FUNCTION "Automatico_linea_1" : VOID	// FC 5
NAME : Auto_L1
VERSION : 0.1
BEGIN
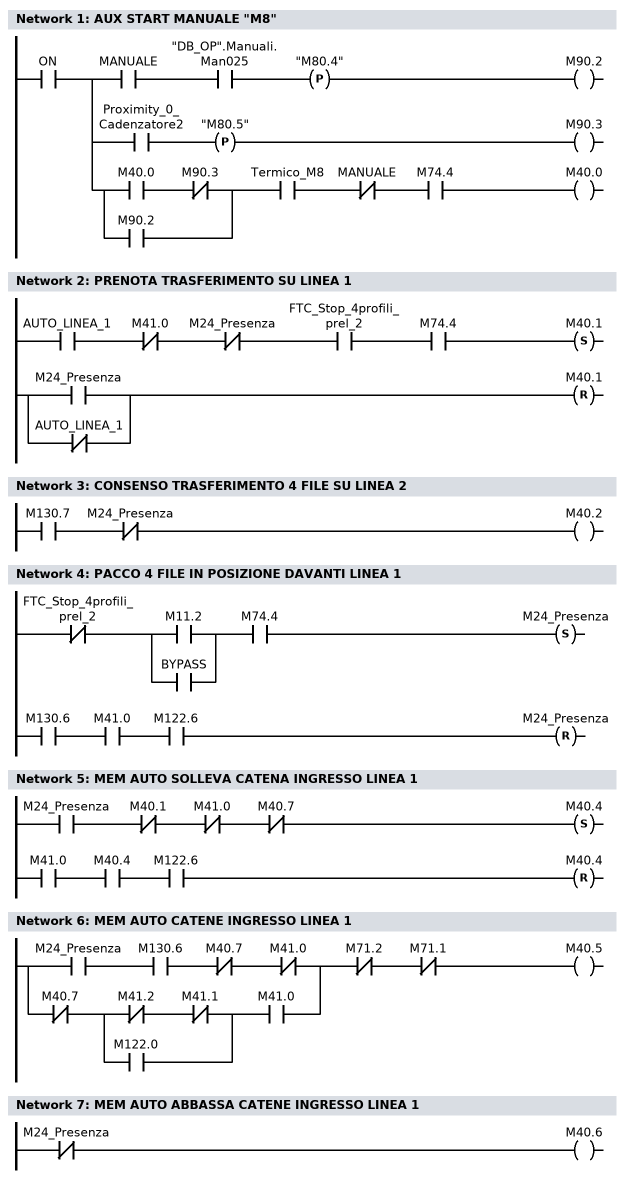
NETWORK
TITLE = AUX START MANUALE "M8"
      A     "ON";
      =     L 0.0;
      A     L 0.0;
      A     "MANUALE";
      A     "DB_OP".Manuali.Man025;
      FP    "M80.4";
      =     "M90.2";
      A     L 0.0;
      A     "Proximity_0_Cadenzatore2";
      FP    "M80.5";
      =     "M90.3";
      A     L 0.0;
      A(;
      A     "M40.0";
      AN    "M90.3";
      O     "M90.2";
      );
      A     "Termico_M8";
      AN    "MANUALE";
      A     "M74.4";
      =     "M40.0";
NETWORK
TITLE = PRENOTA TRASFERIMENTO SU LINEA 1
      A     "AUTO_LINEA_1";
      AN    "M41.0";
      AN    "M24_Presenza";
      A     "FTC_Stop_4profili_prel_2";
      A     "M74.4";
      S     "M40.1";
      A(;
      O     "M24_Presenza";
      ON    "AUTO_LINEA_1";
      );
      R     "M40.1";
      NOP   0;
NETWORK
TITLE = CONSENSO TRASFERIMENTO 4 FILE SU LINEA 2
      A     "M130.7";
      AN    "M24_Presenza";
      =     "M40.2";
NETWORK
TITLE = PACCO 4 FILE IN POSIZIONE DAVANTI LINEA 1
      AN    "FTC_Stop_4profili_prel_2";
      A(;
      O     "M11.2";
      O     "BYPASS";
      );
      A     "M74.4";
      S     "M24_Presenza";
      A     "M130.6";
      A     "M41.0";
      A     "M122.6";
      R     "M24_Presenza";
      NOP   0;
NETWORK
TITLE = MEM AUTO SOLLEVA CATENA INGRESSO LINEA 1
      A     "M24_Presenza";
      AN    "M40.1";
      AN    "M41.0";
      AN    "M40.7";
      S     "M40.4";
      A     "M41.0";
      A     "M40.4";
      A     "M122.6";
      R     "M40.4";
      NOP   0;
NETWORK
TITLE = MEM AUTO CATENE INGRESSO LINEA 1
      A(;
      A     "M24_Presenza";
      A     "M130.6";
      AN    "M40.7";
      AN    "M41.0";
      O;
      AN    "M40.7";
      A(;
      AN    "M41.2";
      AN    "M41.1";
      O     "M122.0";
      );
      A     "M41.0";
      );
      AN    "M71.2";
      AN    "M71.1";
      =     "M40.5";
NETWORK
TITLE = MEM AUTO ABBASSA CATENE INGRESSO LINEA 1
      AN    "M24_Presenza";
      =     "M40.6";
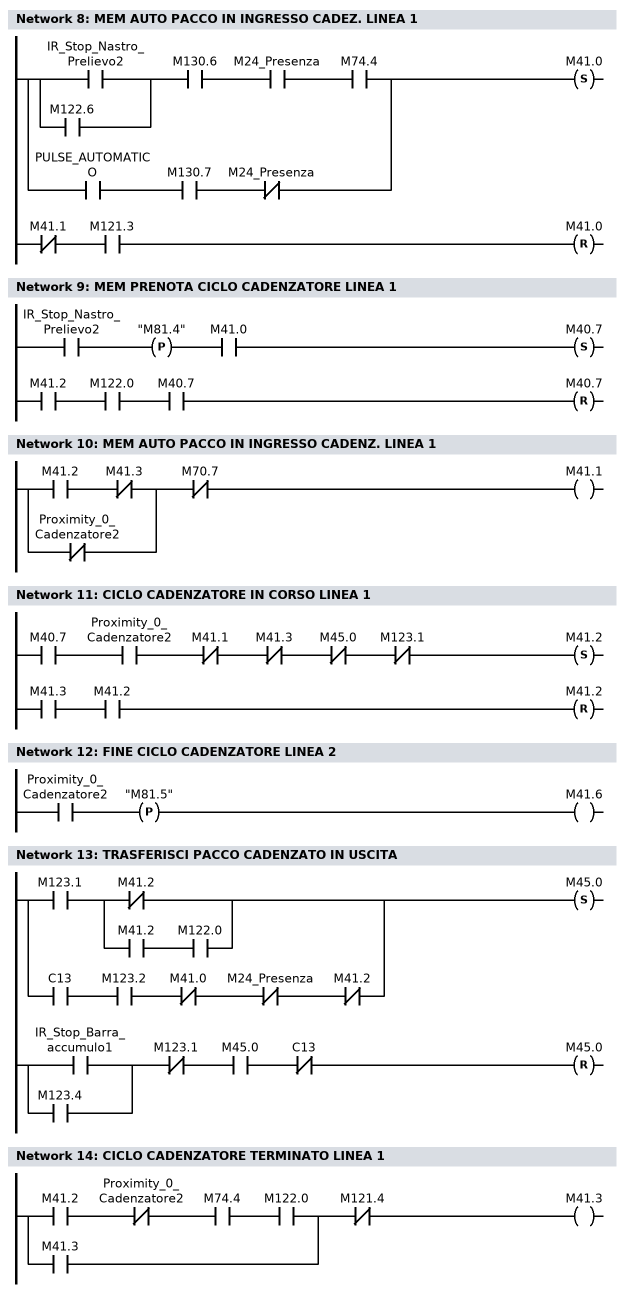
NETWORK
TITLE = MEM AUTO PACCO IN INGRESSO CADEZ. LINEA 1
      A(;
      A(;
      O     "IR_Stop_Nastro_Prelievo2";
      O     "M122.6";
      );
      A     "M130.6";
      A     "M24_Presenza";
      A     "M74.4";
      O;
      A     "PULSE_AUTOMATICO";
      A     "M130.7";
      AN    "M24_Presenza";
      );
      S     "M41.0";
      AN    "M41.1";
      A     "M121.3";
      R     "M41.0";
      NOP   0;
NETWORK
TITLE = MEM PRENOTA CICLO CADENZATORE LINEA 1
      A     "IR_Stop_Nastro_Prelievo2";
      FP    "M81.4";
      A     "M41.0";
      S     "M40.7";
      A     "M41.2";
      A     "M122.0";
      A     "M40.7";
      R     "M40.7";
      NOP   0;
NETWORK
TITLE = MEM AUTO PACCO IN INGRESSO CADENZ. LINEA 1
      A(;
      A     "M41.2";
      AN    "M41.3";
      ON    "Proximity_0_Cadenzatore2";
      );
      AN    "M70.7";
      =     "M41.1";
NETWORK
TITLE = CICLO CADENZATORE IN CORSO LINEA 1
      A     "M40.7";
      A     "Proximity_0_Cadenzatore2";
      AN    "M41.1";
      AN    "M41.3";
      AN    "M45.0";
      AN    "M123.1";
      S     "M41.2";
      A     "M41.3";
      A     "M41.2";
      R     "M41.2";
      NOP   0;
NETWORK
TITLE = FINE CICLO CADENZATORE LINEA 2
      A     "Proximity_0_Cadenzatore2";
      FP    "M81.5";
      =     "M41.6";
NETWORK
TITLE = TRASFERISCI PACCO CADENZATO IN USCITA
      A(;
      A     "M123.1";
      A(;
      ON    "M41.2";
      O;
      A     "M41.2";
      A     "M122.0";
      );
      O;
      A     "C13";
      A     "M123.2";
      AN    "M41.0";
      AN    "M24_Presenza";
      AN    "M41.2";
      );
      S     "M45.0";
      A(;
      O     "IR_Stop_Barra_accumulo1";
      O     "M123.4";
      );
      AN    "M123.1";
      A     "M45.0";
      AN    "C13";
      R     "M45.0";
      NOP   0;
NETWORK
TITLE = CICLO CADENZATORE TERMINATO LINEA 1
      A(;
      A     "M41.2";
      AN    "Proximity_0_Cadenzatore2";
      A     "M74.4";
      A     "M122.0";
      O     "M41.3";
      );
      AN    "M121.4";
      =     "M41.3";
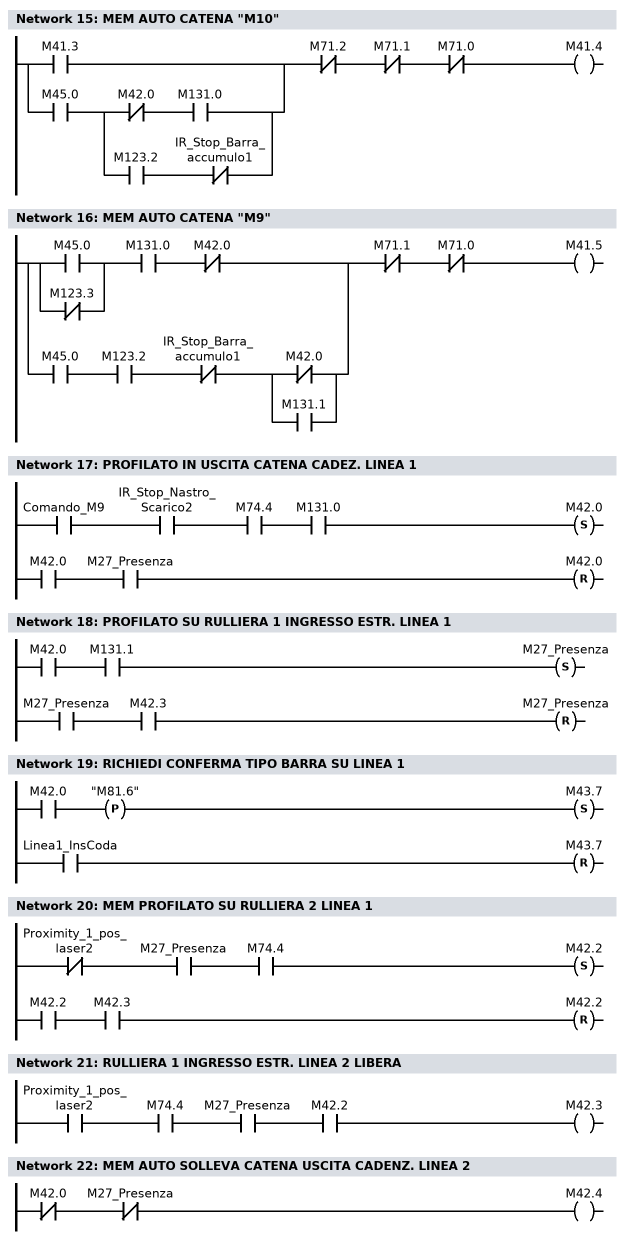
NETWORK
TITLE = MEM AUTO CATENA "M10"
      A(;
      O     "M41.3";
      O;
      A     "M45.0";
      A(;
      AN    "M42.0";
      A     "M131.0";
      O;
      A     "M123.2";
      AN    "IR_Stop_Barra_accumulo1";
      );
      );
      AN    "M71.2";
      AN    "M71.1";
      AN    "M71.0";
      =     "M41.4";
NETWORK
TITLE = MEM AUTO CATENA "M9"
      A(;
      A(;
      O     "M45.0";
      ON    "M123.3";
      );
      A     "M131.0";
      AN    "M42.0";
      O;
      A     "M45.0";
      A     "M123.2";
      AN    "IR_Stop_Barra_accumulo1";
      A(;
      ON    "M42.0";
      O     "M131.1";
      );
      );
      AN    "M71.1";
      AN    "M71.0";
      =     "M41.5";
NETWORK
TITLE = PROFILATO IN USCITA CATENA CADEZ. LINEA 1
      A     "Comando_M9";
      A     "IR_Stop_Nastro_Scarico2";
      A     "M74.4";
      A     "M131.0";
      S     "M42.0";
      A     "M42.0";
      A     "M27_Presenza";
      R     "M42.0";
      NOP   0;
NETWORK
TITLE = PROFILATO SU RULLIERA 1 INGRESSO ESTR. LINEA 1
      A     "M42.0";
      A     "M131.1";
      S     "M27_Presenza";
      A     "M27_Presenza";
      A     "M42.3";
      R     "M27_Presenza";
      NOP   0;
NETWORK
TITLE = RICHIEDI CONFERMA TIPO BARRA SU LINEA 1
      A     "M42.0";
      FP    "M81.6";
      S     "M43.7";
      A     "Linea1_InsCoda";
      R     "M43.7";
      NOP   0;
NETWORK
TITLE = MEM PROFILATO SU RULLIERA 2 LINEA 1
      AN    "Proximity_1_pos_laser2";
      A     "M27_Presenza";
      A     "M74.4";
      S     "M42.2";
      A     "M42.2";
      A     "M42.3";
      R     "M42.2";
      NOP   0;
NETWORK
TITLE = RULLIERA 1 INGRESSO ESTR. LINEA 2 LIBERA
      A     "Proximity_1_pos_laser2";
      A     "M74.4";
      A     "M27_Presenza";
      A     "M42.2";
      =     "M42.3";
NETWORK
TITLE = MEM AUTO SOLLEVA CATENA USCITA CADENZ. LINEA 2
      AN    "M42.0";
      AN    "M27_Presenza";
      =     "M42.4";
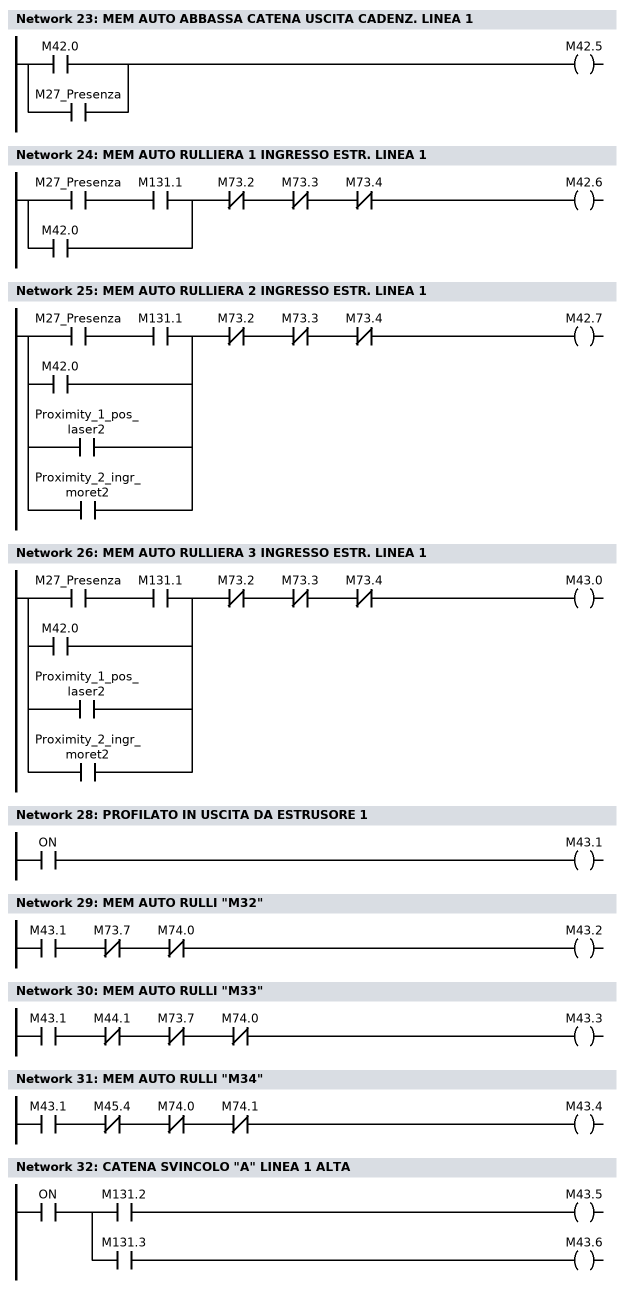
NETWORK
TITLE = MEM AUTO ABBASSA CATENA USCITA CADENZ. LINEA 1
      O     "M42.0";
      O     "M27_Presenza";
      =     "M42.5";
NETWORK
TITLE = MEM AUTO RULLIERA 1 INGRESSO ESTR. LINEA 1
      A(;
      A     "M27_Presenza";
      A     "M131.1";
      O     "M42.0";
      );
      AN    "M73.2";
      AN    "M73.3";
      AN    "M73.4";
      =     "M42.6";
NETWORK
TITLE = MEM AUTO RULLIERA 2 INGRESSO ESTR. LINEA 1
      A(;
      A     "M27_Presenza";
      A     "M131.1";
      O     "M42.0";
      O     "Proximity_1_pos_laser2";
      O     "Proximity_2_ingr_moret2";
      );
      AN    "M73.2";
      AN    "M73.3";
      AN    "M73.4";
      =     "M42.7";
NETWORK
TITLE = MEM AUTO RULLIERA 3 INGRESSO ESTR. LINEA 1
      A(;
      A     "M27_Presenza";
      A     "M131.1";
      O     "M42.0";
      O     "Proximity_1_pos_laser2";
      O     "Proximity_2_ingr_moret2";
      );
      AN    "M73.2";
      AN    "M73.3";
      AN    "M73.4";
      =     "M43.0";
NETWORK
TITLE =
NETWORK
TITLE = PROFILATO IN USCITA DA ESTRUSORE 1
      A     "ON";
      =     "M43.1";
NETWORK
TITLE = MEM AUTO RULLI "M32"
      A     "M43.1";
      AN    "M73.7";
      AN    "M74.0";
      =     "M43.2";
NETWORK
TITLE = MEM AUTO RULLI "M33"
      A     "M43.1";
      AN    "M44.1";
      AN    "M73.7";
      AN    "M74.0";
      =     "M43.3";
NETWORK
TITLE = MEM AUTO RULLI "M34"
      A     "M43.1";
      AN    "M45.4";
      AN    "M74.0";
      AN    "M74.1";
      =     "M43.4";
NETWORK
TITLE = CATENA SVINCOLO "A" LINEA 1 ALTA
      A     "ON";
      =     L 0.0;
      A     L 0.0;
      A     "M131.2";
      =     "M43.5";
      A     L 0.0;
      A     "M131.3";
      =     "M43.6";
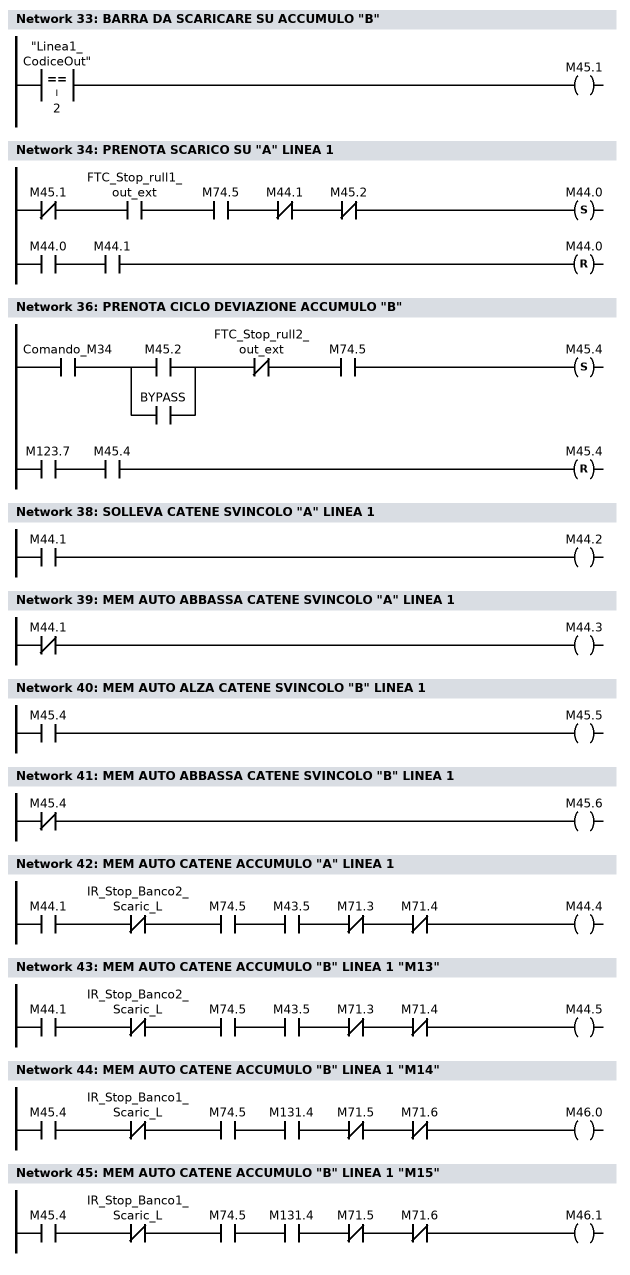
NETWORK
TITLE = BARRA DA SCARICARE SU ACCUMULO "B"
      L     "Linea1_CodiceOut";
      L     2;
      ==I;
      =     "M45.1";
NETWORK
TITLE = PRENOTA SCARICO SU "A" LINEA 1
      AN    "M45.1";
      A     "FTC_Stop_rull1_out_ext";
      A     "M74.5";
      AN    "M44.1";
      AN    "M45.2";
      S     "M44.0";
      A     "M44.0";
      A     "M44.1";
      R     "M44.0";
      NOP   0;
NETWORK
TITLE = SPOSTA BARRA SU RULLIERA "M34"
      A(;
      A     "M45.1";
      AN    "FTC_Stop_rull1_out_ext";
      A     "M74.5";
      AN    "M44.1";
      A     "M43.6";
      S     "M45.2";
      A     "M45.4";
      A     "M45.2";
      R     "M45.2";
      A     "M45.2";
      );
      FP    "M82.2";
      S     "Linea1_DelCoda";
NETWORK
TITLE = PRENOTA CICLO DEVIAZIONE ACCUMULO "B"
      A     "Comando_M34";
      A(;
      O     "M45.2";
      O     "BYPASS";
      );
      AN    "FTC_Stop_rull2_out_ext";
      A     "M74.5";
      S     "M45.4";
      A     "M123.7";
      A     "M45.4";
      R     "M45.4";
      NOP   0;
NETWORK
TITLE = CARICA SU SCARICO "A" LINEA 1
      A(;
      A(;
      AN    "FTC_Stop_rull1_out_ext";
      L     S5T#100MS;
      SD    "T123";
      NOP   0;
      NOP   0;
      NOP   0;
      A     "T123";
      );
      A     "Comando_M33";
      A     "M44.0";
      A     "M74.5";
      A     "M43.6";
      S     "M44.1";
      A     "M123.5";
      A     "M44.1";
      R     "M44.1";
      A     "M44.1";
      );
      FP    "M82.3";
      S     "Linea1_DelCoda";
NETWORK
TITLE = SOLLEVA CATENE SVINCOLO "A" LINEA 1
      A     "M44.1";
      =     "M44.2";
NETWORK
TITLE = MEM AUTO ABBASSA CATENE SVINCOLO "A" LINEA 1
      AN    "M44.1";
      =     "M44.3";
NETWORK
TITLE = MEM AUTO ALZA CATENE SVINCOLO "B" LINEA 1
      A     "M45.4";
      =     "M45.5";
NETWORK
TITLE = MEM AUTO ABBASSA CATENE SVINCOLO "B" LINEA 1
      AN    "M45.4";
      =     "M45.6";
NETWORK
TITLE = MEM AUTO CATENE ACCUMULO "A" LINEA 1
      A     "M44.1";
      AN    "IR_Stop_Banco2_Scaric_L";
      A     "M74.5";
      A     "M43.5";
      AN    "M71.3";
      AN    "M71.4";
      =     "M44.4";
NETWORK
TITLE = MEM AUTO CATENE ACCUMULO "B" LINEA 1 "M13"
      A     "M44.1";
      AN    "IR_Stop_Banco2_Scaric_L";
      A     "M74.5";
      A     "M43.5";
      AN    "M71.3";
      AN    "M71.4";
      =     "M44.5";
NETWORK
TITLE = MEM AUTO CATENE ACCUMULO "B" LINEA 1 "M14"
      A     "M45.4";
      AN    "IR_Stop_Banco1_Scaric_L";
      A     "M74.5";
      A     "M131.4";
      AN    "M71.5";
      AN    "M71.6";
      =     "M46.0";
NETWORK
TITLE = MEM AUTO CATENE ACCUMULO "B" LINEA 1 "M15"
      A     "M45.4";
      AN    "IR_Stop_Banco1_Scaric_L";
      A     "M74.5";
      A     "M131.4";
      AN    "M71.5";
      AN    "M71.6";
      =     "M46.1";
END_FUNCTION

FUNCTION "Automatico_linea_2" : VOID	// FC 6
NAME : Auto_L2
VERSION : 0.1
BEGIN
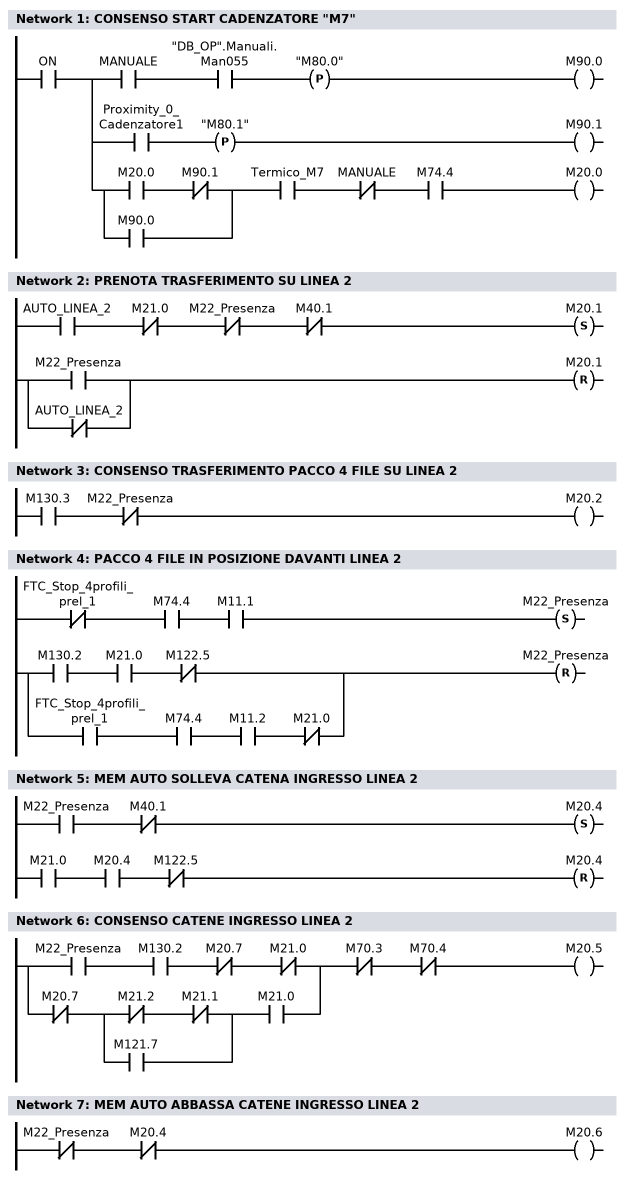
NETWORK
TITLE = CONSENSO START CADENZATORE "M7"
      A     "ON";
      =     L 0.0;
      A     L 0.0;
      A     "MANUALE";
      A     "DB_OP".Manuali.Man055;
      FP    "M80.0";
      =     "M90.0";
      A     L 0.0;
      A     "Proximity_0_Cadenzatore1";
      FP    "M80.1";
      =     "M90.1";
      A     L 0.0;
      A(;
      A     "M20.0";
      AN    "M90.1";
      O     "M90.0";
      );
      A     "Termico_M7";
      AN    "MANUALE";
      A     "M74.4";
      =     "M20.0";
NETWORK
TITLE = PRENOTA TRASFERIMENTO SU LINEA 2
      A     "AUTO_LINEA_2";
      AN    "M21.0";
      AN    "M22_Presenza";
      AN    "M40.1";
      S     "M20.1";
      A(;
      O     "M22_Presenza";
      ON    "AUTO_LINEA_2";
      );
      R     "M20.1";
      NOP   0;
NETWORK
TITLE = CONSENSO TRASFERIMENTO PACCO 4 FILE SU LINEA 2
      A     "M130.3";
      AN    "M22_Presenza";
      =     "M20.2";
NETWORK
TITLE = PACCO 4 FILE IN POSIZIONE DAVANTI LINEA 2
      AN    "FTC_Stop_4profili_prel_1";
      A     "M74.4";
      A     "M11.1";
      S     "M22_Presenza";
      A(;
      A     "M130.2";
      A     "M21.0";
      AN    "M122.5";
      O;
      A     "FTC_Stop_4profili_prel_1";
      A     "M74.4";
      A     "M11.2";
      AN    "M21.0";
      );
      R     "M22_Presenza";
      NOP   0;
NETWORK
TITLE = MEM AUTO SOLLEVA CATENA INGRESSO LINEA 2
      A     "M22_Presenza";
      AN    "M40.1";
      S     "M20.4";
      A     "M21.0";
      A     "M20.4";
      AN    "M122.5";
      R     "M20.4";
      NOP   0;
NETWORK
TITLE = CONSENSO CATENE INGRESSO LINEA 2
      A(;
      A     "M22_Presenza";
      A     "M130.2";
      AN    "M20.7";
      AN    "M21.0";
      O;
      AN    "M20.7";
      A(;
      AN    "M21.2";
      AN    "M21.1";
      O     "M121.7";
      );
      A     "M21.0";
      );
      AN    "M70.3";
      AN    "M70.4";
      =     "M20.5";
NETWORK
TITLE = MEM AUTO ABBASSA CATENE INGRESSO LINEA 2
      AN    "M22_Presenza";
      AN    "M20.4";
      =     "M20.6";
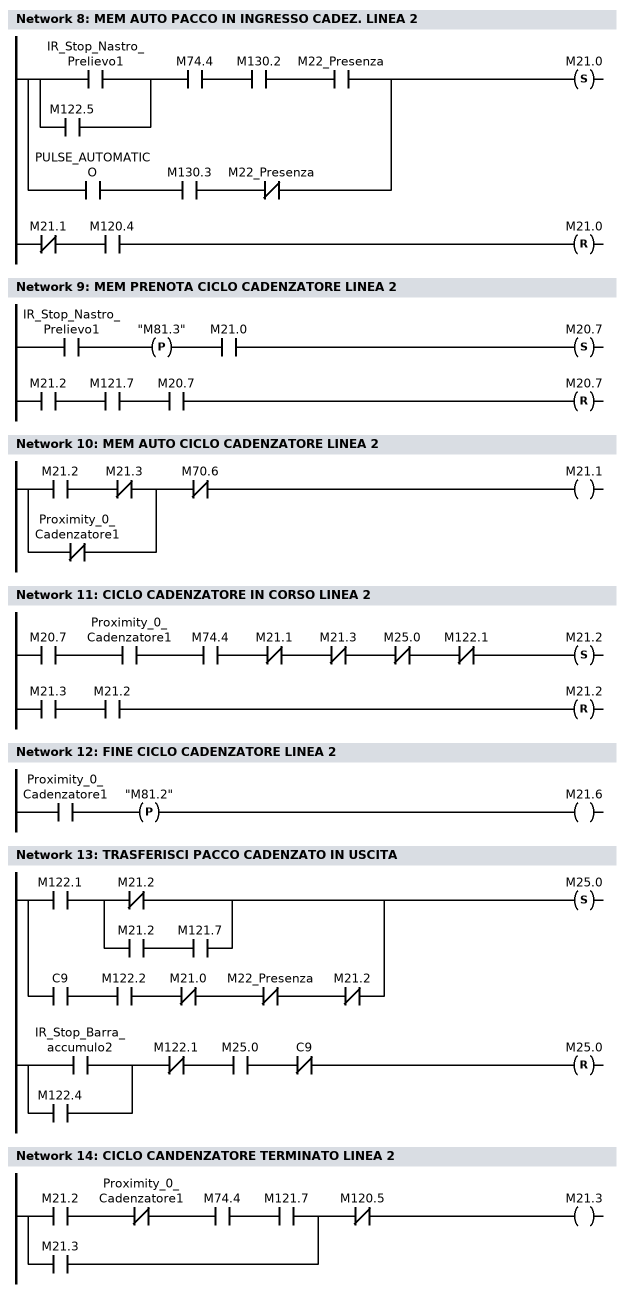
NETWORK
TITLE = MEM AUTO PACCO IN INGRESSO CADEZ. LINEA 2
      A(;
      A(;
      O     "IR_Stop_Nastro_Prelievo1";
      O     "M122.5";
      );
      A     "M74.4";
      A     "M130.2";
      A     "M22_Presenza";
      O;
      A     "PULSE_AUTOMATICO";
      A     "M130.3";
      AN    "M22_Presenza";
      );
      S     "M21.0";
      AN    "M21.1";
      A     "M120.4";
      R     "M21.0";
      NOP   0;
NETWORK
TITLE = MEM PRENOTA CICLO CADENZATORE LINEA 2
      A     "IR_Stop_Nastro_Prelievo1";
      FP    "M81.3";
      A     "M21.0";
      S     "M20.7";
      A     "M21.2";
      A     "M121.7";
      A     "M20.7";
      R     "M20.7";
      NOP   0;
NETWORK
TITLE = MEM AUTO CICLO CADENZATORE LINEA 2
      A(;
      A     "M21.2";
      AN    "M21.3";
      ON    "Proximity_0_Cadenzatore1";
      );
      AN    "M70.6";
      =     "M21.1";
NETWORK
TITLE = CICLO CADENZATORE IN CORSO LINEA 2
      A     "M20.7";
      A     "Proximity_0_Cadenzatore1";
      A     "M74.4";
      AN    "M21.1";
      AN    "M21.3";
      AN    "M25.0";
      AN    "M122.1";
      S     "M21.2";
      A     "M21.3";
      A     "M21.2";
      R     "M21.2";
      NOP   0;
NETWORK
TITLE = FINE CICLO CADENZATORE LINEA 2
      A     "Proximity_0_Cadenzatore1";
      FP    "M81.2";
      =     "M21.6";
NETWORK
TITLE = TRASFERISCI PACCO CADENZATO IN USCITA
      A(;
      A     "M122.1";
      A(;
      ON    "M21.2";
      O;
      A     "M21.2";
      A     "M121.7";
      );
      O;
      A     "C9";
      A     "M122.2";
      AN    "M21.0";
      AN    "M22_Presenza";
      AN    "M21.2";
      );
      S     "M25.0";
      A(;
      O     "IR_Stop_Barra_accumulo2";
      O     "M122.4";
      );
      AN    "M122.1";
      A     "M25.0";
      AN    "C9";
      R     "M25.0";
      NOP   0;
NETWORK
TITLE = CICLO CANDENZATORE TERMINATO LINEA 2
      A(;
      A     "M21.2";
      AN    "Proximity_0_Cadenzatore1";
      A     "M74.4";
      A     "M121.7";
      O     "M21.3";
      );
      AN    "M120.5";
      =     "M21.3";
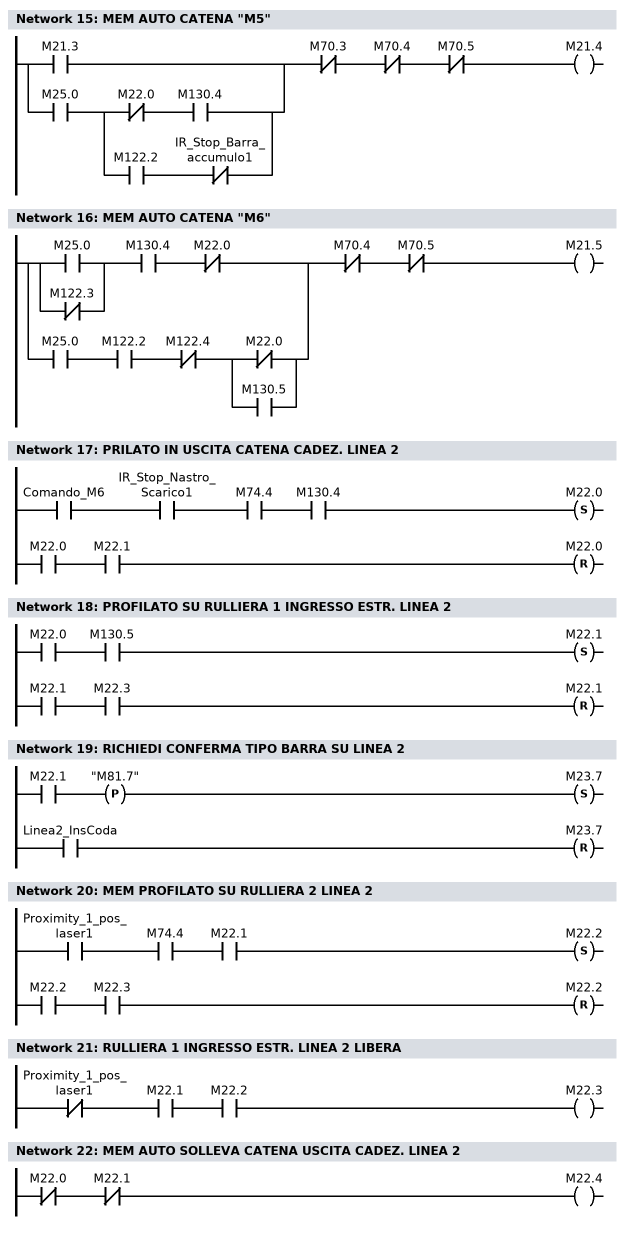
NETWORK
TITLE = MEM AUTO CATENA "M5"
      A(;
      O     "M21.3";
      O;
      A     "M25.0";
      A(;
      AN    "M22.0";
      A     "M130.4";
      O;
      A     "M122.2";
      AN    "IR_Stop_Barra_accumulo1";
      );
      );
      AN    "M70.3";
      AN    "M70.4";
      AN    "M70.5";
      =     "M21.4";
NETWORK
TITLE = MEM AUTO CATENA "M6"
      A(;
      A(;
      O     "M25.0";
      ON    "M122.3";
      );
      A     "M130.4";
      AN    "M22.0";
      O;
      A     "M25.0";
      A     "M122.2";
      AN    "M122.4";
      A(;
      ON    "M22.0";
      O     "M130.5";
      );
      );
      AN    "M70.4";
      AN    "M70.5";
      =     "M21.5";
NETWORK
TITLE = PRILATO IN USCITA CATENA CADEZ. LINEA 2
      A     "Comando_M6";
      A     "IR_Stop_Nastro_Scarico1";
      A     "M74.4";
      A     "M130.4";
      S     "M22.0";
      A     "M22.0";
      A     "M22.1";
      R     "M22.0";
      NOP   0;
NETWORK
TITLE = PROFILATO SU RULLIERA 1 INGRESSO ESTR. LINEA 2
      A     "M22.0";
      A     "M130.5";
      S     "M22.1";
      A     "M22.1";
      A     "M22.3";
      R     "M22.1";
      NOP   0;
NETWORK
TITLE = RICHIEDI CONFERMA TIPO BARRA SU LINEA 2
      A     "M22.1";
      FP    "M81.7";
      S     "M23.7";
      A     "Linea2_InsCoda";
      R     "M23.7";
      NOP   0;
NETWORK
TITLE = MEM PROFILATO SU RULLIERA 2 LINEA 2
      A     "Proximity_1_pos_laser1";
      A     "M74.4";
      A     "M22.1";
      S     "M22.2";
      A     "M22.2";
      A     "M22.3";
      R     "M22.2";
      NOP   0;
NETWORK
TITLE = RULLIERA 1 INGRESSO ESTR. LINEA 2 LIBERA
      AN    "Proximity_1_pos_laser1";
      A     "M22.1";
      A     "M22.2";
      =     "M22.3";
NETWORK
TITLE = MEM AUTO SOLLEVA CATENA USCITA CADEZ. LINEA 2
      AN    "M22.0";
      AN    "M22.1";
      =     "M22.4";
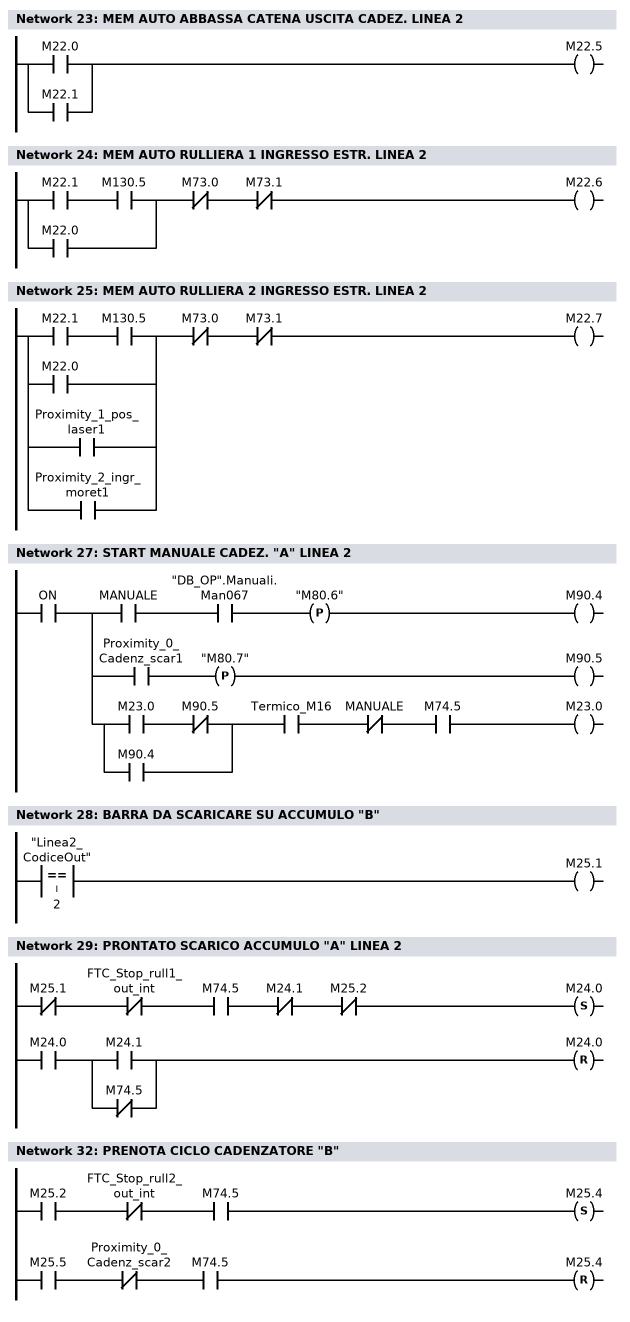
NETWORK
TITLE = MEM AUTO ABBASSA CATENA USCITA CADEZ. LINEA 2
      O     "M22.0";
      O     "M22.1";
      =     "M22.5";
NETWORK
TITLE = MEM AUTO RULLIERA 1 INGRESSO ESTR. LINEA 2
      A(;
      A     "M22.1";
      A     "M130.5";
      O     "M22.0";
      );
      AN    "M73.0";
      AN    "M73.1";
      =     "M22.6";
NETWORK
TITLE = MEM AUTO RULLIERA 2 INGRESSO ESTR. LINEA 2
      A(;
      A     "M22.1";
      A     "M130.5";
      O     "M22.0";
      O     "Proximity_1_pos_laser1";
      O     "Proximity_2_ingr_moret1";
      );
      AN    "M73.0";
      AN    "M73.1";
      =     "M22.7";
NETWORK
TITLE =
NETWORK
TITLE = START MANUALE CADEZ. "A" LINEA 2
      A     "ON";
      =     L 0.0;
      A     L 0.0;
      A     "MANUALE";
      A     "DB_OP".Manuali.Man067;
      FP    "M80.6";
      =     "M90.4";
      A     L 0.0;
      A     "Proximity_0_Cadenz_scar1";
      FP    "M80.7";
      =     "M90.5";
      A     L 0.0;
      A(;
      A     "M23.0";
      AN    "M90.5";
      O     "M90.4";
      );
      A     "Termico_M16";
      AN    "MANUALE";
      A     "M74.5";
      =     "M23.0";
NETWORK
TITLE = BARRA DA SCARICARE SU ACCUMULO "B"
      L     "Linea2_CodiceOut";
      L     2;
      ==I;
      =     "M25.1";
NETWORK
TITLE = PRONTATO SCARICO ACCUMULO "A" LINEA 2
      AN    "M25.1";
      AN    "FTC_Stop_rull1_out_int";
      A     "M74.5";
      AN    "M24.1";
      AN    "M25.2";
      S     "M24.0";
      A     "M24.0";
      A(;
      O     "M24.1";
      ON    "M74.5";
      );
      R     "M24.0";
      NOP   0;
NETWORK
TITLE = SPOSTA BASSA RU RULLIERA "M31"
      A(;
      A     "M25.1";
      AN    "FTC_Stop_rull1_out_int";
      A     "M74.5";
      AN    "M24.1";
      S     "M25.2";
      A     "M25.4";
      A     "M25.2";
      R     "M25.2";
      A     "M25.2";
      );
      FP    "M82.1";
      S     "Linea2_DelCoda";
NETWORK
TITLE = PROFILATO PRONTO SU CADEZ. "A" LINEA 2
      A(;
      A(;
      AN    "FTC_Stop_rull1_out_int";
      L     S5T#100MS;
      SD    "T124";
      NOP   0;
      NOP   0;
      NOP   0;
      A     "T124";
      );
      A     "M24.0";
      A     "M74.5";
      S     "M24.1";
      A     "M24.2";
      AN    "Proximity_0_Cadenz_scar1";
      A     "M74.5";
      R     "M24.1";
      A     "M24.1";
      );
      FP    "M82.0";
      S     "Linea2_DelCoda";
NETWORK
TITLE = PRENOTA CICLO CADENZATORE "B"
      A     "M25.2";
      AN    "FTC_Stop_rull2_out_int";
      A     "M74.5";
      S     "M25.4";
      A     "M25.5";
      AN    "Proximity_0_Cadenz_scar2";
      A     "M74.5";
      R     "M25.4";
      NOP   0;
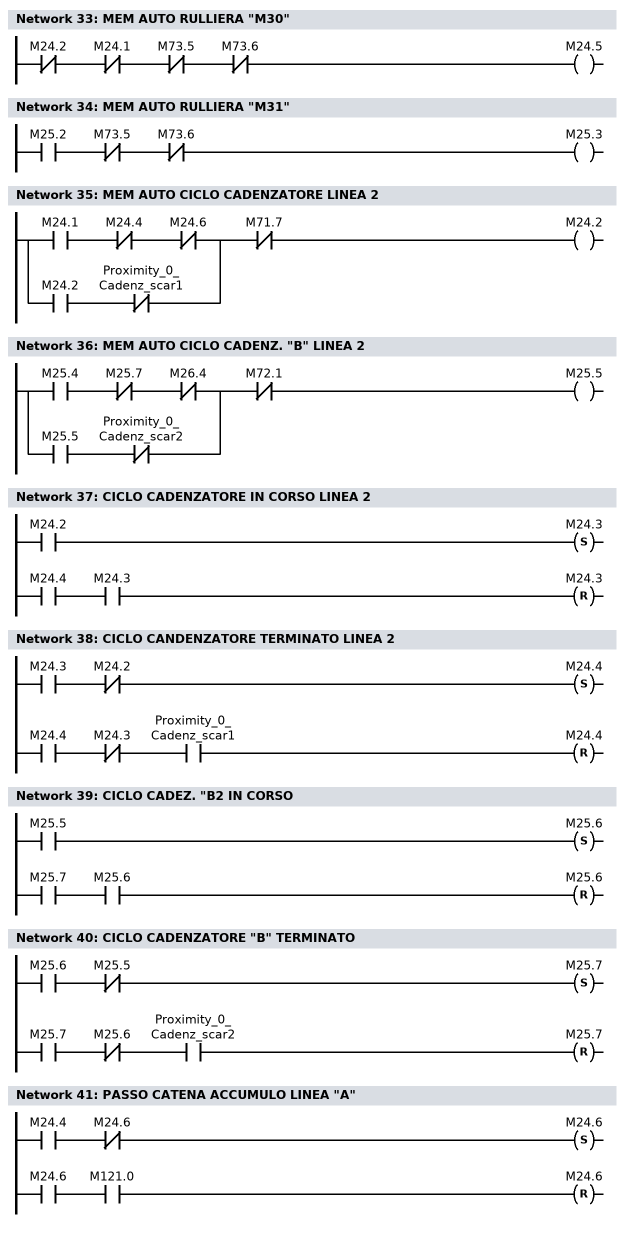
NETWORK
TITLE = MEM AUTO RULLIERA "M30"
      AN    "M24.2";
      AN    "M24.1";
      AN    "M73.5";
      AN    "M73.6";
      =     "M24.5";
NETWORK
TITLE = MEM AUTO RULLIERA "M31"
      A     "M25.2";
      AN    "M73.5";
      AN    "M73.6";
      =     "M25.3";
NETWORK
TITLE = MEM AUTO CICLO CADENZATORE LINEA 2
      A(;
      A     "M24.1";
      AN    "M24.4";
      AN    "M24.6";
      O;
      A     "M24.2";
      AN    "Proximity_0_Cadenz_scar1";
      );
      AN    "M71.7";
      =     "M24.2";
NETWORK
TITLE = MEM AUTO CICLO CADENZ. "B" LINEA 2
      A(;
      A     "M25.4";
      AN    "M25.7";
      AN    "M26.4";
      O;
      A     "M25.5";
      AN    "Proximity_0_Cadenz_scar2";
      );
      AN    "M72.1";
      =     "M25.5";
NETWORK
TITLE = CICLO CADENZATORE IN CORSO LINEA 2
      A     "M24.2";
      S     "M24.3";
      A     "M24.4";
      A     "M24.3";
      R     "M24.3";
      NOP   0;
NETWORK
TITLE = CICLO CANDENZATORE TERMINATO LINEA 2
      A     "M24.3";
      AN    "M24.2";
      S     "M24.4";
      A     "M24.4";
      AN    "M24.3";
      A     "Proximity_0_Cadenz_scar1";
      R     "M24.4";
      NOP   0;
NETWORK
TITLE = CICLO CADEZ. "B2 IN CORSO
      A     "M25.5";
      S     "M25.6";
      A     "M25.7";
      A     "M25.6";
      R     "M25.6";
      NOP   0;
NETWORK
TITLE = CICLO CADENZATORE "B" TERMINATO
      A     "M25.6";
      AN    "M25.5";
      S     "M25.7";
      A     "M25.7";
      AN    "M25.6";
      A     "Proximity_0_Cadenz_scar2";
      R     "M25.7";
      NOP   0;
NETWORK
TITLE = PASSO CATENA ACCUMULO LINEA "A"
      A     "M24.4";
      AN    "M24.6";
      S     "M24.6";
      A     "M24.6";
      A     "M121.0";
      R     "M24.6";
      NOP   0;
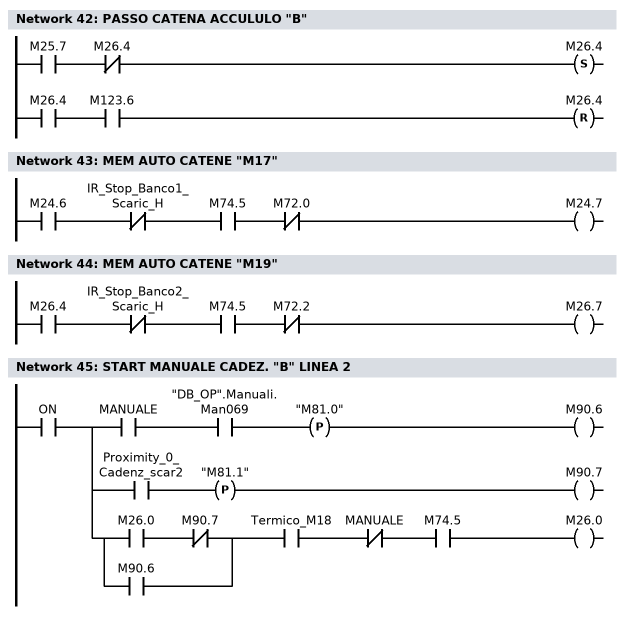
NETWORK
TITLE = PASSO CATENA ACCULULO "B"
      A     "M25.7";
      AN    "M26.4";
      S     "M26.4";
      A     "M26.4";
      A     "M123.6";
      R     "M26.4";
      NOP   0;
NETWORK
TITLE = MEM AUTO CATENE "M17"
      A     "M24.6";
      AN    "IR_Stop_Banco1_Scaric_H";
      A     "M74.5";
      AN    "M72.0";
      =     "M24.7";
NETWORK
TITLE = MEM AUTO CATENE "M19"
      A     "M26.4";
      AN    "IR_Stop_Banco2_Scaric_H";
      A     "M74.5";
      AN    "M72.2";
      =     "M26.7";
NETWORK
TITLE = START MANUALE CADEZ. "B" LINEA 2
      A     "ON";
      =     L 0.0;
      A     L 0.0;
      A     "MANUALE";
      A     "DB_OP".Manuali.Man069;
      FP    "M81.0";
      =     "M90.6";
      A     L 0.0;
      A     "Proximity_0_Cadenz_scar2";
      FP    "M81.1";
      =     "M90.7";
      A     L 0.0;
      A(;
      A     "M26.0";
      AN    "M90.7";
      O     "M90.6";
      );
      A     "Termico_M18";
      AN    "MANUALE";
      A     "M74.5";
      =     "M26.0";
END_FUNCTION

FUNCTION "PROFIBUS_MM4" : VOID	// FC 10
AUTHOR : PROTEKNO
NAME : MM4
VERSION : 0.1
VAR_INPUT
  Periferic_Address : INT ;
  Drive_On_Off : BOOL ;
  Drive_Reversing : BOOL ;
  Drive_Fault_ACKN : BOOL ;
  Drive_F_Setpoint : REAL ;
END_VAR
VAR_OUTPUT
  Drive_in_operation : BOOL ;
  Drive_Fault_Active : BOOL ;
  Drive_Alarm_Active : BOOL ;
  Freno : BOOL ;
  Drive_F_Act : REAL ;
END_VAR
VAR_TEMP
  Address_E_A : DWORD ;
  SEND : STRUCT
   CW1 : UDT 1;
   f_setpoint : WORD ;
  END_STRUCT ;
  REC : STRUCT
   SW1 : UDT 2;
   f_act : WORD ;
  END_STRUCT ;
END_VAR
BEGIN
NETWORK
TITLE = Trasferimento indirizzo blocco;
      L     #Periferic_Address;
      SLD   3;
      T     #Address_E_A;
NETWORK
TITLE = Status word PZD MM4;
      L     PID [#Address_E_A];
      T     #REC;	//Status word MM4;
NETWORK
TITLE = control bit`s + setpoint
// ---------------------------------------
// IN-Variablen FC
// --------------------------------------
// PZD1 - Steuerwort 1                  // set single bit in the control word 1
      SET;	// set VKE=1
      =     #SEND.CW1.Bit_1;
      =     #SEND.CW1.Bit_2;
      =     #SEND.CW1.Bit_3;
      =     #SEND.CW1.Bit_4;
      =     #SEND.CW1.Bit_5;
      =     #SEND.CW1.Bit_6;
      =     #SEND.CW1.Bit_10;	// setpoint valid
      CLR;	// set VKE=0
      =     #SEND.CW1.Bit_8;
      =     #SEND.CW1.Bit_9;
      =     #SEND.CW1.Bit_12;
      =     #SEND.CW1.Bit_13;
      =     #SEND.CW1.Bit_14;
      =     #SEND.CW1.Bit_15;
      A     #Drive_On_Off;	// on / off ?
      =     #SEND.CW1.Bit_0;
      A     #Drive_Reversing;	// cw / cww ?
      =     #SEND.CW1.Bit_11;
      A     #Drive_Fault_ACKN;	// fault ackn.?
      =     #SEND.CW1.Bit_7;
//  
// PZD2 - Drehzahlsollwert
// gültiger Drehzahlsollwert zwischen 0.00-50 Hz
      L     #Drive_F_Setpoint;	// setpoint [Hz]
      L     0.000000e+00;
      <R;	// setpoinz >0Hz
      JC    N004;
      L     #Drive_F_Setpoint;
      L     7.500000e+01;
      >R;	// setpoint < 75Hz ?
      JC    N004;
      L     #Drive_F_Setpoint;
      L     1.000000e+02;	// 2-Nachkommastellen retten
      *R;
      RND;	//conversion of a 32-bit IEEE floating-point number to 32-bit integer
      L     24576;	// 16384 = 4000HEX = 50Hz
      *D;
      L     7500;
      /D;
      T     #SEND.f_setpoint;
N004: NOP   0;
NETWORK
TITLE = stateword + actual frequency 
// -------------------------------------
// OUT-Variablen FC                     
// -------------------------------------
// PZD 1 - Zustandswort
      A     #REC.SW1.Bit_2;
      =     #Drive_in_operation;
      A     #REC.SW1.Bit_3;
      =     #Drive_Fault_Active;
      A     #REC.SW1.Bit_7;
      =     #Drive_Alarm_Active;
      A     #REC.SW1.Bit_12;
      =     #Freno;
// PZD 2 - Drehzahlistwert
      L     #REC.f_act;
      ITD;
      DTR;
      L     5.000000e+01;	//16383= 4000HEX = 50Hz
      *R;
      L     1.638400e+04;
      /R;
      L     1.000000e+02;
      *R;
      TRUNC;
      ITD;
      DTR;
      L     1.000000e+02;
      /R;
      T     #Drive_F_Act;
NETWORK
TITLE = Control word PZD MM4;
      L     #SEND;	//Control word MM4;
      T     PQD [#Address_E_A];
      BE;
END_FUNCTION

FUNCTION "Comandi_zona_ingresso" : VOID	// FC 14
VERSION : 0.1
BEGIN
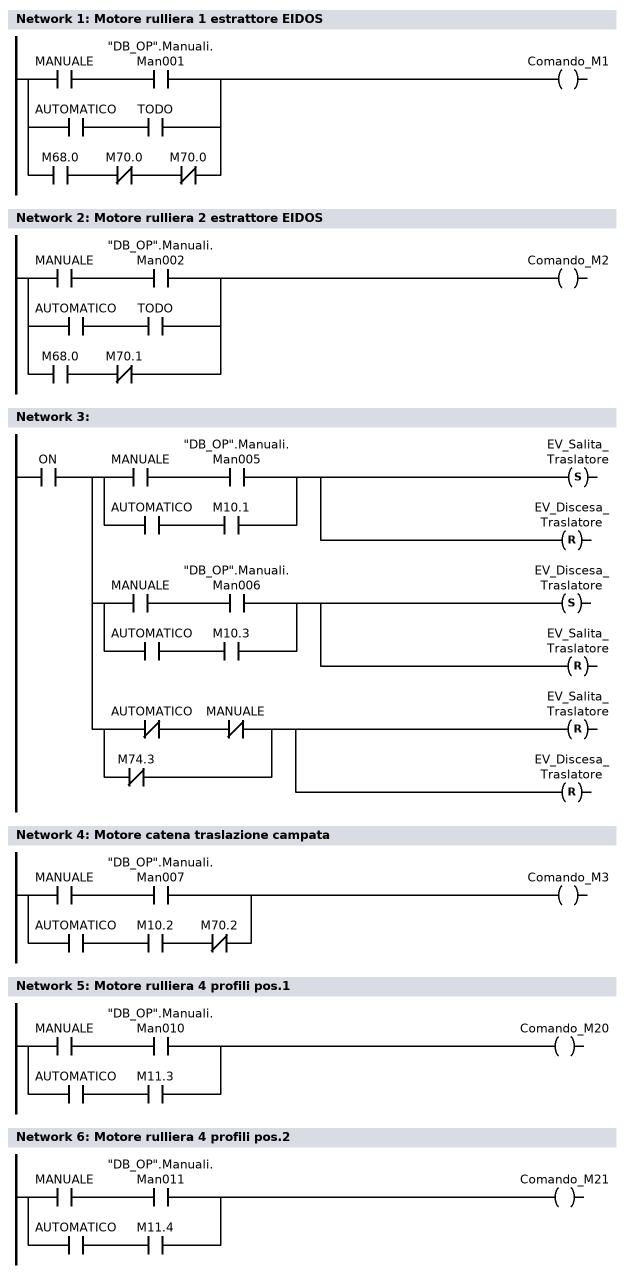
NETWORK
TITLE = Motore rulliera 1 estrattore EIDOS
      A     "MANUALE";
      A     "DB_OP".Manuali.Man001;
      O;
      A     "AUTOMATICO";
      A     "TODO";
      O;
      A     "M68.0";
      AN    "M70.0";
      AN    "M70.0";
      =     "Comando_M1";
NETWORK
TITLE = Motore rulliera 2 estrattore EIDOS
      A     "MANUALE";
      A     "DB_OP".Manuali.Man002;
      O;
      A     "AUTOMATICO";
      A     "TODO";
      O;
      A     "M68.0";
      AN    "M70.1";
      =     "Comando_M2";
NETWORK
TITLE =
      A     "ON";
      =     L 0.0;
      A     L 0.0;
      A(;
      A     "MANUALE";
      A     "DB_OP".Manuali.Man005;
      O;
      A     "AUTOMATICO";
      A     "M10.1";
      );
      S     "EV_Salita_Traslatore";
      R     "EV_Discesa_Traslatore";
      A     L 0.0;
      A(;
      A     "MANUALE";
      A     "DB_OP".Manuali.Man006;
      O;
      A     "AUTOMATICO";
      A     "M10.3";
      );
      S     "EV_Discesa_Traslatore";
      R     "EV_Salita_Traslatore";
      A     L 0.0;
      A(;
      AN    "AUTOMATICO";
      AN    "MANUALE";
      ON    "M74.3";
      );
      R     "EV_Salita_Traslatore";
      R     "EV_Discesa_Traslatore";
NETWORK
TITLE = Motore catena traslazione campata
      A     "MANUALE";
      A     "DB_OP".Manuali.Man007;
      O;
      A     "AUTOMATICO";
      A     "M10.2";
      AN    "M70.2";
      =     "Comando_M3";
NETWORK
TITLE = Motore rulliera 4 profili pos.1
      A     "MANUALE";
      A     "DB_OP".Manuali.Man010;
      O;
      A     "AUTOMATICO";
      A     "M11.3";
      =     "Comando_M20";
NETWORK
TITLE = Motore rulliera 4 profili pos.2
      A     "MANUALE";
      A     "DB_OP".Manuali.Man011;
      O;
      A     "AUTOMATICO";
      A     "M11.4";
      =     "Comando_M21";
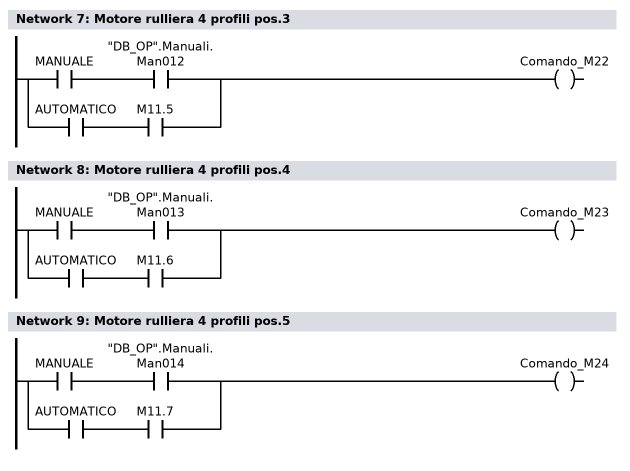
NETWORK
TITLE = Motore rulliera 4 profili pos.3
      A     "MANUALE";
      A     "DB_OP".Manuali.Man012;
      O;
      A     "AUTOMATICO";
      A     "M11.5";
      =     "Comando_M22";
NETWORK
TITLE = Motore rulliera 4 profili pos.4
      A     "MANUALE";
      A     "DB_OP".Manuali.Man013;
      O;
      A     "AUTOMATICO";
      A     "M11.6";
      =     "Comando_M23";
NETWORK
TITLE = Motore rulliera 4 profili pos.5
      A     "MANUALE";
      A     "DB_OP".Manuali.Man014;
      O;
      A     "AUTOMATICO";
      A     "M11.7";
      =     "Comando_M24";
END_FUNCTION

FUNCTION "Comandi_linea_1" : VOID	// FC 15
VERSION : 0.1
BEGIN
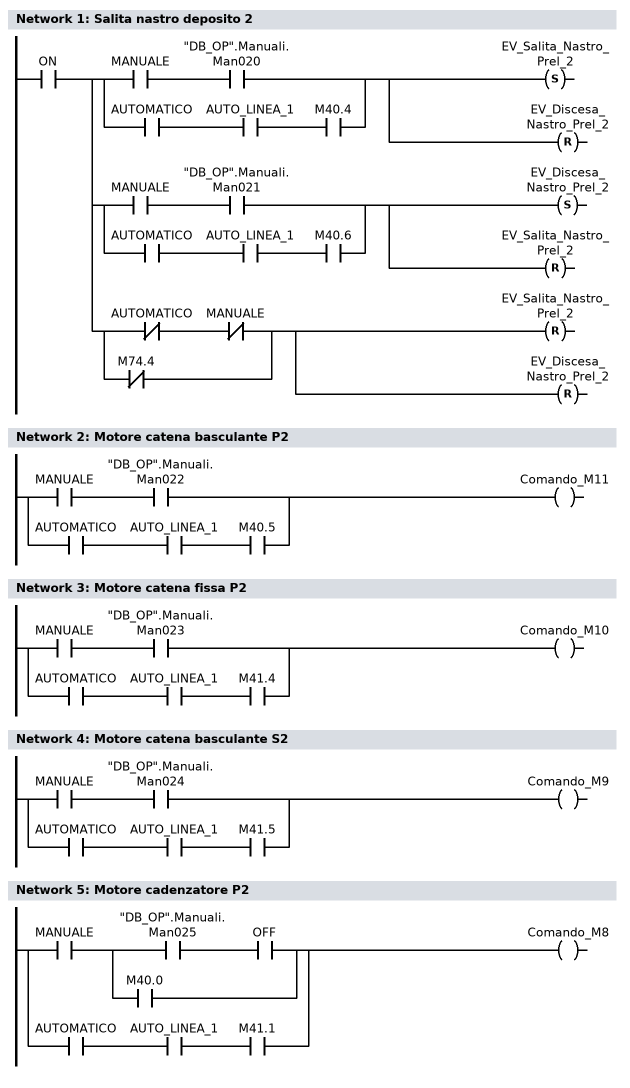
NETWORK
TITLE = Salita nastro deposito 2
      A     "ON";
      =     L 0.0;
      A     L 0.0;
      A(;
      A     "MANUALE";
      A     "DB_OP".Manuali.Man020;
      O;
      A     "AUTOMATICO";
      A     "AUTO_LINEA_1";
      A     "M40.4";
      );
      S     "EV_Salita_Nastro_Prel_2";
      R     "EV_Discesa_Nastro_Prel_2";
      A     L 0.0;
      A(;
      A     "MANUALE";
      A     "DB_OP".Manuali.Man021;
      O;
      A     "AUTOMATICO";
      A     "AUTO_LINEA_1";
      A     "M40.6";
      );
      S     "EV_Discesa_Nastro_Prel_2";
      R     "EV_Salita_Nastro_Prel_2";
      A     L 0.0;
      A(;
      AN    "AUTOMATICO";
      AN    "MANUALE";
      ON    "M74.4";
      );
      R     "EV_Salita_Nastro_Prel_2";
      R     "EV_Discesa_Nastro_Prel_2";
NETWORK
TITLE = Motore catena basculante P2
      A     "MANUALE";
      A     "DB_OP".Manuali.Man022;
      O;
      A     "AUTOMATICO";
      A     "AUTO_LINEA_1";
      A     "M40.5";
      =     "Comando_M11";
NETWORK
TITLE = Motore catena fissa P2
      A     "MANUALE";
      A     "DB_OP".Manuali.Man023;
      O;
      A     "AUTOMATICO";
      A     "AUTO_LINEA_1";
      A     "M41.4";
      =     "Comando_M10";
NETWORK
TITLE = Motore catena basculante S2
      A     "MANUALE";
      A     "DB_OP".Manuali.Man024;
      O;
      A     "AUTOMATICO";
      A     "AUTO_LINEA_1";
      A     "M41.5";
      =     "Comando_M9";
NETWORK
TITLE = Motore cadenzatore P2
      A     "MANUALE";
      A(;
      A     "DB_OP".Manuali.Man025;
      A     "OFF";
      O     "M40.0";
      );
      O;
      A     "AUTOMATICO";
      A     "AUTO_LINEA_1";
      A     "M41.1";
      =     "Comando_M8";
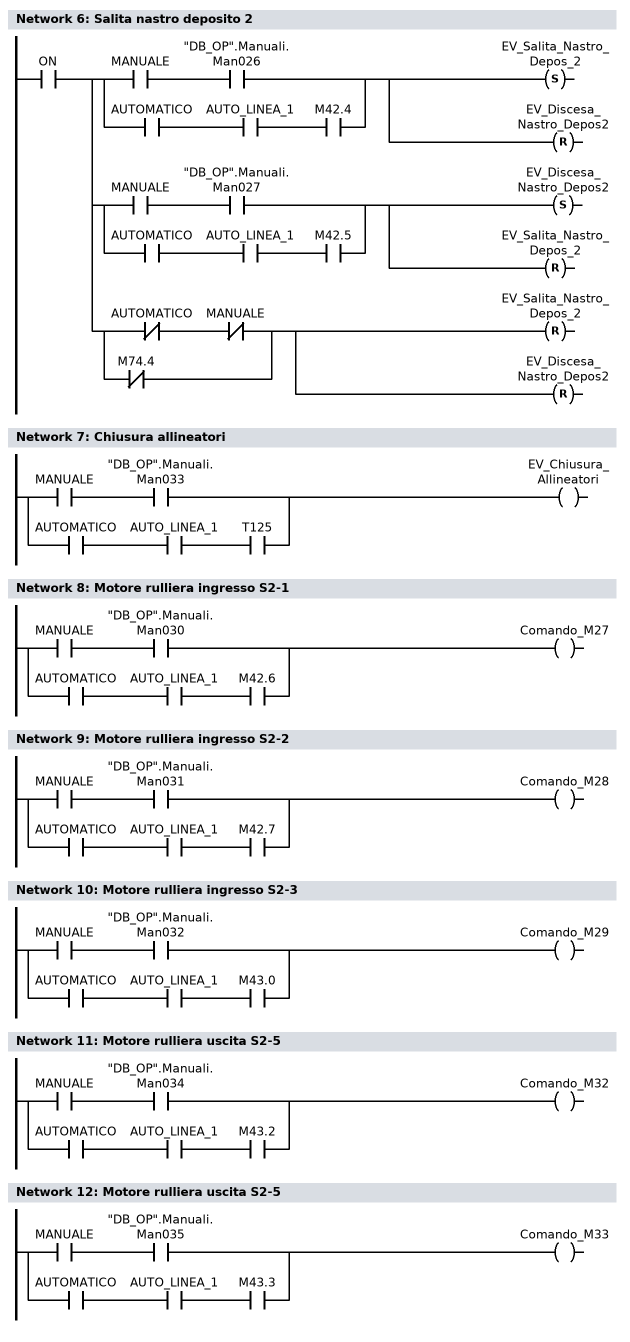
NETWORK
TITLE = Salita nastro deposito 2
      A     "ON";
      =     L 0.0;
      A     L 0.0;
      A(;
      A     "MANUALE";
      A     "DB_OP".Manuali.Man026;
      O;
      A     "AUTOMATICO";
      A     "AUTO_LINEA_1";
      A     "M42.4";
      );
      S     "EV_Salita_Nastro_Depos_2";
      R     "EV_Discesa_Nastro_Depos2";
      A     L 0.0;
      A(;
      A     "MANUALE";
      A     "DB_OP".Manuali.Man027;
      O;
      A     "AUTOMATICO";
      A     "AUTO_LINEA_1";
      A     "M42.5";
      );
      S     "EV_Discesa_Nastro_Depos2";
      R     "EV_Salita_Nastro_Depos_2";
      A     L 0.0;
      A(;
      AN    "AUTOMATICO";
      AN    "MANUALE";
      ON    "M74.4";
      );
      R     "EV_Salita_Nastro_Depos_2";
      R     "EV_Discesa_Nastro_Depos2";
NETWORK
TITLE = Chiusura allineatori
      A     "MANUALE";
      A     "DB_OP".Manuali.Man033;
      O;
      A     "AUTOMATICO";
      A     "AUTO_LINEA_1";
      A     "T125";
      =     "EV_Chiusura_Allineatori";
NETWORK
TITLE = Motore rulliera ingresso S2-1
      A     "MANUALE";
      A     "DB_OP".Manuali.Man030;
      O;
      A     "AUTOMATICO";
      A     "AUTO_LINEA_1";
      A     "M42.6";
      =     "Comando_M27";
NETWORK
TITLE = Motore rulliera ingresso S2-2
      A     "MANUALE";
      A     "DB_OP".Manuali.Man031;
      O;
      A     "AUTOMATICO";
      A     "AUTO_LINEA_1";
      A     "M42.7";
      =     "Comando_M28";
NETWORK
TITLE = Motore rulliera ingresso S2-3
      A     "MANUALE";
      A     "DB_OP".Manuali.Man032;
      O;
      A     "AUTOMATICO";
      A     "AUTO_LINEA_1";
      A     "M43.0";
      =     "Comando_M29";
NETWORK
TITLE = Motore rulliera uscita S2-5
      A     "MANUALE";
      A     "DB_OP".Manuali.Man034;
      O;
      A     "AUTOMATICO";
      A     "AUTO_LINEA_1";
      A     "M43.2";
      =     "Comando_M32";
NETWORK
TITLE = Motore rulliera uscita S2-5
      A     "MANUALE";
      A     "DB_OP".Manuali.Man035;
      O;
      A     "AUTOMATICO";
      A     "AUTO_LINEA_1";
      A     "M43.3";
      =     "Comando_M33";
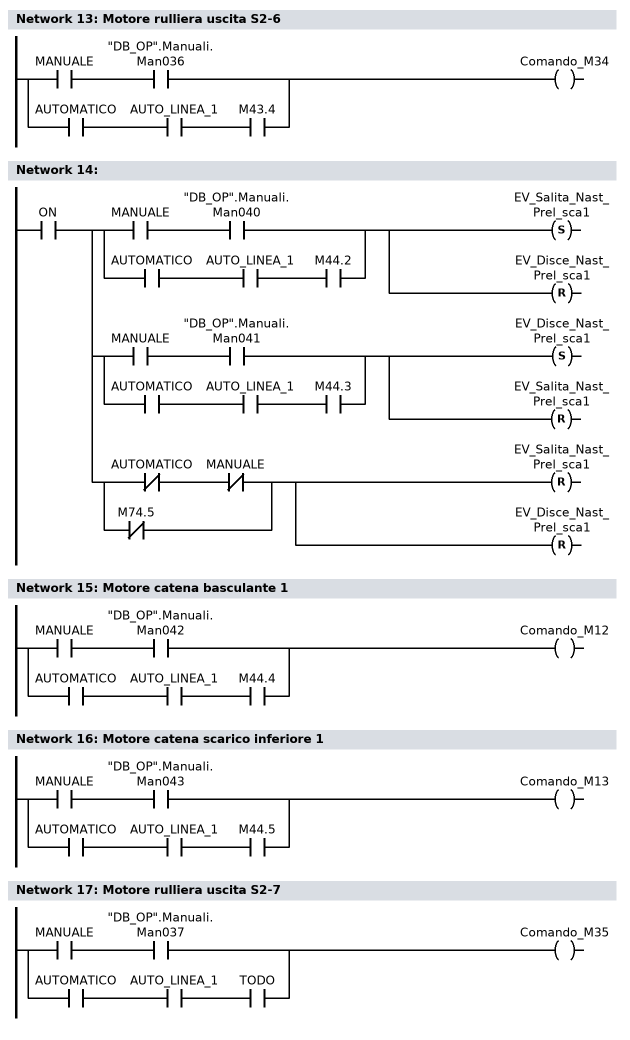
NETWORK
TITLE = Motore rulliera uscita S2-6
      A     "MANUALE";
      A     "DB_OP".Manuali.Man036;
      O;
      A     "AUTOMATICO";
      A     "AUTO_LINEA_1";
      A     "M43.4";
      =     "Comando_M34";
NETWORK
TITLE =
      A     "ON";
      =     L 0.0;
      A     L 0.0;
      A(;
      A     "MANUALE";
      A     "DB_OP".Manuali.Man040;
      O;
      A     "AUTOMATICO";
      A     "AUTO_LINEA_1";
      A     "M44.2";
      );
      S     "EV_Salita_Nast_Prel_sca1";
      R     "EV_Disce_Nast_Prel_sca1";
      A     L 0.0;
      A(;
      A     "MANUALE";
      A     "DB_OP".Manuali.Man041;
      O;
      A     "AUTOMATICO";
      A     "AUTO_LINEA_1";
      A     "M44.3";
      );
      S     "EV_Disce_Nast_Prel_sca1";
      R     "EV_Salita_Nast_Prel_sca1";
      A     L 0.0;
      A(;
      AN    "AUTOMATICO";
      AN    "MANUALE";
      ON    "M74.5";
      );
      R     "EV_Salita_Nast_Prel_sca1";
      R     "EV_Disce_Nast_Prel_sca1";
NETWORK
TITLE = Motore catena basculante 1
      A     "MANUALE";
      A     "DB_OP".Manuali.Man042;
      O;
      A     "AUTOMATICO";
      A     "AUTO_LINEA_1";
      A     "M44.4";
      =     "Comando_M12";
NETWORK
TITLE = Motore catena scarico inferiore 1
      A     "MANUALE";
      A     "DB_OP".Manuali.Man043;
      O;
      A     "AUTOMATICO";
      A     "AUTO_LINEA_1";
      A     "M44.5";
      =     "Comando_M13";
NETWORK
TITLE = Motore rulliera uscita S2-7
      A     "MANUALE";
      A     "DB_OP".Manuali.Man037;
      O;
      A     "AUTOMATICO";
      A     "AUTO_LINEA_1";
      A     "TODO";
      =     "Comando_M35";
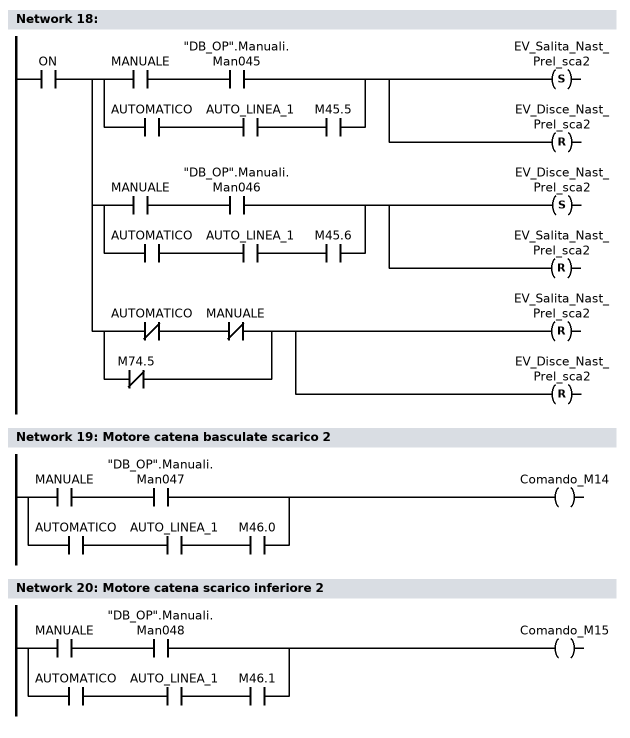
NETWORK
TITLE =
      A     "ON";
      =     L 0.0;
      A     L 0.0;
      A(;
      A     "MANUALE";
      A     "DB_OP".Manuali.Man045;
      O;
      A     "AUTOMATICO";
      A     "AUTO_LINEA_1";
      A     "M45.5";
      );
      S     "EV_Salita_Nast_Prel_sca2";
      R     "EV_Disce_Nast_Prel_sca2";
      A     L 0.0;
      A(;
      A     "MANUALE";
      A     "DB_OP".Manuali.Man046;
      O;
      A     "AUTOMATICO";
      A     "AUTO_LINEA_1";
      A     "M45.6";
      );
      S     "EV_Disce_Nast_Prel_sca2";
      R     "EV_Salita_Nast_Prel_sca2";
      A     L 0.0;
      A(;
      AN    "AUTOMATICO";
      AN    "MANUALE";
      ON    "M74.5";
      );
      R     "EV_Salita_Nast_Prel_sca2";
      R     "EV_Disce_Nast_Prel_sca2";
NETWORK
TITLE = Motore catena basculate scarico 2
      A     "MANUALE";
      A     "DB_OP".Manuali.Man047;
      O;
      A     "AUTOMATICO";
      A     "AUTO_LINEA_1";
      A     "M46.0";
      =     "Comando_M14";
NETWORK
TITLE = Motore catena scarico inferiore 2
      A     "MANUALE";
      A     "DB_OP".Manuali.Man048;
      O;
      A     "AUTOMATICO";
      A     "AUTO_LINEA_1";
      A     "M46.1";
      =     "Comando_M15";
END_FUNCTION

FUNCTION "Comandi_linea_2" : VOID	// FC 16
VERSION : 0.1
BEGIN
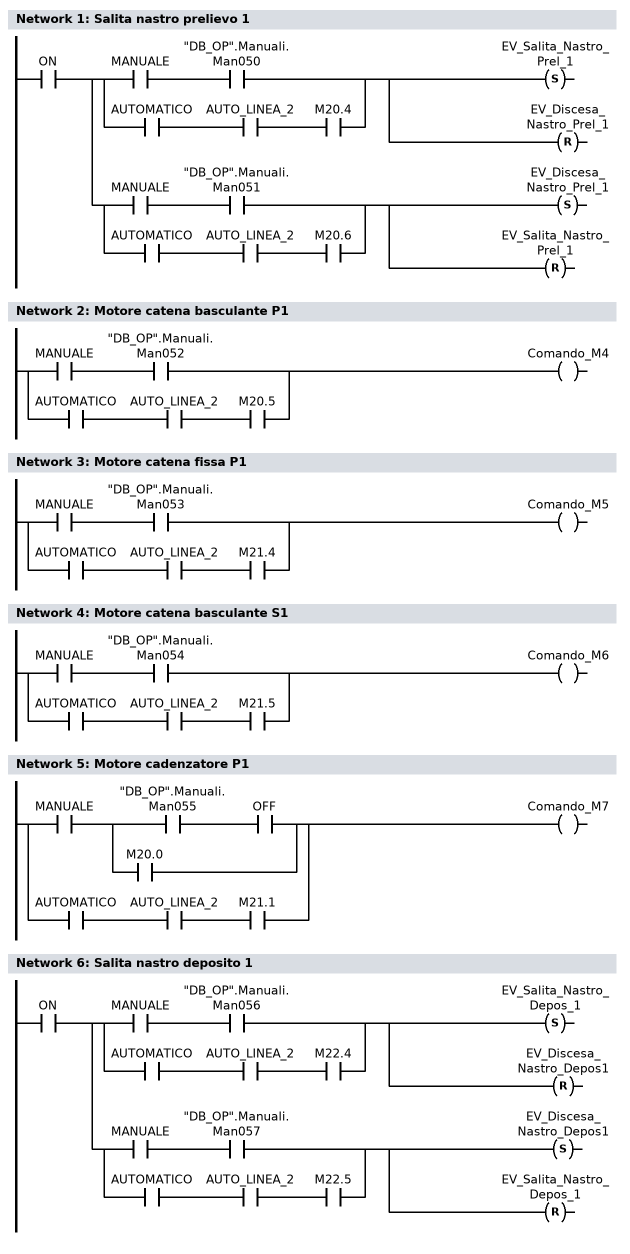
NETWORK
TITLE = Salita nastro prelievo 1
      A     "ON";
      =     L 0.0;
      A     L 0.0;
      A(;
      A     "MANUALE";
      A     "DB_OP".Manuali.Man050;
      O;
      A     "AUTOMATICO";
      A     "AUTO_LINEA_2";
      A     "M20.4";
      );
      S     "EV_Salita_Nastro_Prel_1";
      R     "EV_Discesa_Nastro_Prel_1";
      A     L 0.0;
      A(;
      A     "MANUALE";
      A     "DB_OP".Manuali.Man051;
      O;
      A     "AUTOMATICO";
      A     "AUTO_LINEA_2";
      A     "M20.6";
      );
      S     "EV_Discesa_Nastro_Prel_1";
      R     "EV_Salita_Nastro_Prel_1";
NETWORK
TITLE = Motore catena basculante P1
      A     "MANUALE";
      A     "DB_OP".Manuali.Man052;
      O;
      A     "AUTOMATICO";
      A     "AUTO_LINEA_2";
      A     "M20.5";
      =     "Comando_M4";
NETWORK
TITLE = Motore catena fissa P1
      A     "MANUALE";
      A     "DB_OP".Manuali.Man053;
      O;
      A     "AUTOMATICO";
      A     "AUTO_LINEA_2";
      A     "M21.4";
      =     "Comando_M5";
NETWORK
TITLE = Motore catena basculante S1
      A     "MANUALE";
      A     "DB_OP".Manuali.Man054;
      O;
      A     "AUTOMATICO";
      A     "AUTO_LINEA_2";
      A     "M21.5";
      =     "Comando_M6";
NETWORK
TITLE = Motore cadenzatore P1
      A     "MANUALE";
      A(;
      A     "DB_OP".Manuali.Man055;
      A     "OFF";
      O     "M20.0";
      );
      O;
      A     "AUTOMATICO";
      A     "AUTO_LINEA_2";
      A     "M21.1";
      =     "Comando_M7";
NETWORK
TITLE = Salita nastro deposito 1
      A     "ON";
      =     L 0.0;
      A     L 0.0;
      A(;
      A     "MANUALE";
      A     "DB_OP".Manuali.Man056;
      O;
      A     "AUTOMATICO";
      A     "AUTO_LINEA_2";
      A     "M22.4";
      );
      S     "EV_Salita_Nastro_Depos_1";
      R     "EV_Discesa_Nastro_Depos1";
      A     L 0.0;
      A(;
      A     "MANUALE";
      A     "DB_OP".Manuali.Man057;
      O;
      A     "AUTOMATICO";
      A     "AUTO_LINEA_2";
      A     "M22.5";
      );
      S     "EV_Discesa_Nastro_Depos1";
      R     "EV_Salita_Nastro_Depos_1";
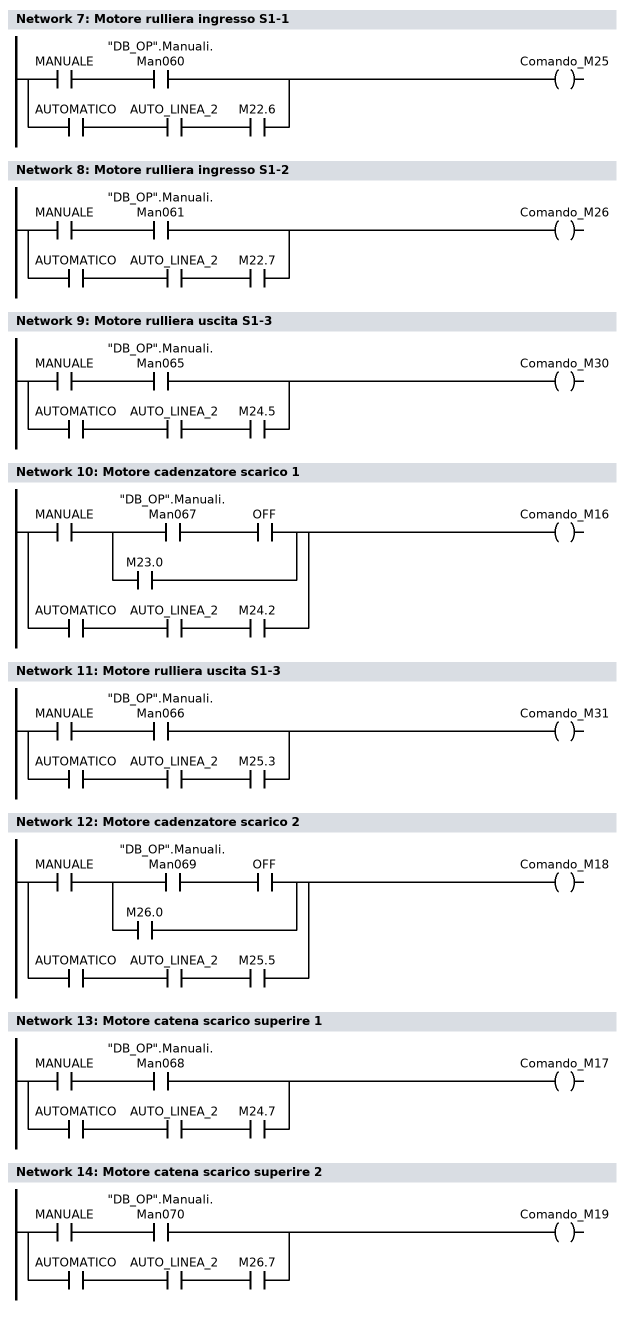
NETWORK
TITLE = Motore rulliera ingresso S1-1
      A     "MANUALE";
      A     "DB_OP".Manuali.Man060;
      O;
      A     "AUTOMATICO";
      A     "AUTO_LINEA_2";
      A     "M22.6";
      =     "Comando_M25";
NETWORK
TITLE = Motore rulliera ingresso S1-2
      A     "MANUALE";
      A     "DB_OP".Manuali.Man061;
      O;
      A     "AUTOMATICO";
      A     "AUTO_LINEA_2";
      A     "M22.7";
      =     "Comando_M26";
NETWORK
TITLE = Motore rulliera uscita S1-3
      A     "MANUALE";
      A     "DB_OP".Manuali.Man065;
      O;
      A     "AUTOMATICO";
      A     "AUTO_LINEA_2";
      A     "M24.5";
      =     "Comando_M30";
NETWORK
TITLE = Motore cadenzatore scarico 1
      A     "MANUALE";
      A(;
      A     "DB_OP".Manuali.Man067;
      A     "OFF";
      O     "M23.0";
      );
      O;
      A     "AUTOMATICO";
      A     "AUTO_LINEA_2";
      A     "M24.2";
      =     "Comando_M16";
NETWORK
TITLE = Motore rulliera uscita S1-3
      A     "MANUALE";
      A     "DB_OP".Manuali.Man066;
      O;
      A     "AUTOMATICO";
      A     "AUTO_LINEA_2";
      A     "M25.3";
      =     "Comando_M31";
NETWORK
TITLE = Motore cadenzatore scarico 2
      A     "MANUALE";
      A(;
      A     "DB_OP".Manuali.Man069;
      A     "OFF";
      O     "M26.0";
      );
      O;
      A     "AUTOMATICO";
      A     "AUTO_LINEA_2";
      A     "M25.5";
      =     "Comando_M18";
NETWORK
TITLE = Motore catena scarico superire 1
      A     "MANUALE";
      A     "DB_OP".Manuali.Man068;
      O;
      A     "AUTOMATICO";
      A     "AUTO_LINEA_2";
      A     "M24.7";
      =     "Comando_M17";
NETWORK
TITLE = Motore catena scarico superire 2
      A     "MANUALE";
      A     "DB_OP".Manuali.Man070;
      O;
      A     "AUTOMATICO";
      A     "AUTO_LINEA_2";
      A     "M26.7";
      =     "Comando_M19";
END_FUNCTION

FUNCTION "Comandi_Inverter" : VOID	// FC 17
VERSION : 0.1
VAR_TEMP
  Temp1 : BOOL ;
  Temp2 : BOOL ;
  Temp3 : BOOL ;
  Temp4 : BOOL ;
  RTemp1 : REAL ;
END_VAR
BEGIN
NETWORK
TITLE =
      CALL  "PROFIBUS_MM4" (
           Periferic_Address        := 280,
           Drive_On_Off             := "Comando_M20",
           Drive_Reversing          := FALSE,
           Drive_Fault_ACKN         := FALSE,
           Drive_F_Setpoint         := 7.000000e+01,
           Drive_in_operation       := #Temp1,
           Drive_Fault_Active       := "M66.0",
           Drive_Alarm_Active       := #Temp3,
           Freno                    := #Temp4,
           Drive_F_Act              := #RTemp1);
NETWORK
TITLE =
      CALL  "PROFIBUS_MM4" (
           Periferic_Address        := 292,
           Drive_On_Off             := "Comando_M21",
           Drive_Reversing          := FALSE,
           Drive_Fault_ACKN         := FALSE,
           Drive_F_Setpoint         := 7.000000e+01,
           Drive_in_operation       := #Temp1,
           Drive_Fault_Active       := "M66.1",
           Drive_Alarm_Active       := #Temp3,
           Freno                    := #Temp4,
           Drive_F_Act              := #RTemp1);
NETWORK
TITLE =
      CALL  "PROFIBUS_MM4" (
           Periferic_Address        := 304,
           Drive_On_Off             := "Comando_M22",
           Drive_Reversing          := FALSE,
           Drive_Fault_ACKN         := FALSE,
           Drive_F_Setpoint         := 7.000000e+01,
           Drive_in_operation       := #Temp1,
           Drive_Fault_Active       := "M66.2",
           Drive_Alarm_Active       := #Temp3,
           Freno                    := #Temp4,
           Drive_F_Act              := #RTemp1);
NETWORK
TITLE =
      CALL  "PROFIBUS_MM4" (
           Periferic_Address        := 316,
           Drive_On_Off             := "Comando_M23",
           Drive_Reversing          := FALSE,
           Drive_Fault_ACKN         := FALSE,
           Drive_F_Setpoint         := 7.000000e+01,
           Drive_in_operation       := #Temp1,
           Drive_Fault_Active       := "M66.3",
           Drive_Alarm_Active       := #Temp3,
           Freno                    := #Temp4,
           Drive_F_Act              := #RTemp1);
NETWORK
TITLE =
      CALL  "PROFIBUS_MM4" (
           Periferic_Address        := 328,
           Drive_On_Off             := "Comando_M24",
           Drive_Reversing          := FALSE,
           Drive_Fault_ACKN         := FALSE,
           Drive_F_Setpoint         := 7.000000e+01,
           Drive_in_operation       := #Temp1,
           Drive_Fault_Active       := "M66.4",
           Drive_Alarm_Active       := #Temp3,
           Freno                    := #Temp4,
           Drive_F_Act              := #RTemp1);
NETWORK
TITLE =
      CALL  "PROFIBUS_MM4" (
           Periferic_Address        := 340,
           Drive_On_Off             := "Comando_M25",
           Drive_Reversing          := FALSE,
           Drive_Fault_ACKN         := FALSE,
           Drive_F_Setpoint         := 5.000000e+01,
           Drive_in_operation       := #Temp1,
           Drive_Fault_Active       := "M66.5",
           Drive_Alarm_Active       := #Temp3,
           Freno                    := #Temp4,
           Drive_F_Act              := #RTemp1);
NETWORK
TITLE =
      CALL  "PROFIBUS_MM4" (
           Periferic_Address        := 352,
           Drive_On_Off             := "Comando_M26",
           Drive_Reversing          := FALSE,
           Drive_Fault_ACKN         := FALSE,
           Drive_F_Setpoint         := 5.000000e+01,
           Drive_in_operation       := #Temp1,
           Drive_Fault_Active       := "M66.6",
           Drive_Alarm_Active       := #Temp3,
           Freno                    := #Temp4,
           Drive_F_Act              := #RTemp1);
NETWORK
TITLE =
      CALL  "PROFIBUS_MM4" (
           Periferic_Address        := 364,
           Drive_On_Off             := "Comando_M27",
           Drive_Reversing          := FALSE,
           Drive_Fault_ACKN         := FALSE,
           Drive_F_Setpoint         := 5.000000e+01,
           Drive_in_operation       := #Temp1,
           Drive_Fault_Active       := "M66.7",
           Drive_Alarm_Active       := #Temp3,
           Freno                    := #Temp4,
           Drive_F_Act              := #RTemp1);
NETWORK
TITLE =
      CALL  "PROFIBUS_MM4" (
           Periferic_Address        := 376,
           Drive_On_Off             := "Comando_M28",
           Drive_Reversing          := FALSE,
           Drive_Fault_ACKN         := FALSE,
           Drive_F_Setpoint         := 5.000000e+01,
           Drive_in_operation       := #Temp1,
           Drive_Fault_Active       := "M67.0",
           Drive_Alarm_Active       := #Temp3,
           Freno                    := #Temp4,
           Drive_F_Act              := #RTemp1);
NETWORK
TITLE =
      CALL  "PROFIBUS_MM4" (
           Periferic_Address        := 388,
           Drive_On_Off             := "Comando_M29",
           Drive_Reversing          := FALSE,
           Drive_Fault_ACKN         := FALSE,
           Drive_F_Setpoint         := 5.000000e+01,
           Drive_in_operation       := #Temp1,
           Drive_Fault_Active       := "M67.1",
           Drive_Alarm_Active       := #Temp3,
           Freno                    := #Temp4,
           Drive_F_Act              := #RTemp1);
NETWORK
TITLE =
      CALL  "PROFIBUS_MM4" (
           Periferic_Address        := 400,
           Drive_On_Off             := "Comando_M30",
           Drive_Reversing          := FALSE,
           Drive_Fault_ACKN         := FALSE,
           Drive_F_Setpoint         := 5.000000e+01,
           Drive_in_operation       := #Temp1,
           Drive_Fault_Active       := "M67.2",
           Drive_Alarm_Active       := #Temp3,
           Freno                    := #Temp4,
           Drive_F_Act              := #RTemp1);
NETWORK
TITLE =
      CALL  "PROFIBUS_MM4" (
           Periferic_Address        := 412,
           Drive_On_Off             := "Comando_M31",
           Drive_Reversing          := FALSE,
           Drive_Fault_ACKN         := FALSE,
           Drive_F_Setpoint         := 5.000000e+01,
           Drive_in_operation       := #Temp1,
           Drive_Fault_Active       := "M67.3",
           Drive_Alarm_Active       := #Temp3,
           Freno                    := #Temp4,
           Drive_F_Act              := #RTemp1);
NETWORK
TITLE =
      CALL  "PROFIBUS_MM4" (
           Periferic_Address        := 424,
           Drive_On_Off             := "Comando_M32",
           Drive_Reversing          := FALSE,
           Drive_Fault_ACKN         := FALSE,
           Drive_F_Setpoint         := 5.000000e+01,
           Drive_in_operation       := #Temp1,
           Drive_Fault_Active       := "M67.4",
           Drive_Alarm_Active       := #Temp3,
           Freno                    := #Temp4,
           Drive_F_Act              := #RTemp1);
NETWORK
TITLE =
      CALL  "PROFIBUS_MM4" (
           Periferic_Address        := 436,
           Drive_On_Off             := "Comando_M33",
           Drive_Reversing          := FALSE,
           Drive_Fault_ACKN         := FALSE,
           Drive_F_Setpoint         := 5.000000e+01,
           Drive_in_operation       := #Temp1,
           Drive_Fault_Active       := "M67.5",
           Drive_Alarm_Active       := #Temp3,
           Freno                    := #Temp4,
           Drive_F_Act              := #RTemp1);
NETWORK
TITLE =
      CALL  "PROFIBUS_MM4" (
           Periferic_Address        := 448,
           Drive_On_Off             := "Comando_M34",
           Drive_Reversing          := FALSE,
           Drive_Fault_ACKN         := FALSE,
           Drive_F_Setpoint         := 5.000000e+01,
           Drive_in_operation       := #Temp1,
           Drive_Fault_Active       := "M67.6",
           Drive_Alarm_Active       := #Temp3,
           Freno                    := #Temp4,
           Drive_F_Act              := #RTemp1);
NETWORK
TITLE =
      CALL  "PROFIBUS_MM4" (
           Periferic_Address        := 460,
           Drive_On_Off             := "Comando_M35",
           Drive_Reversing          := FALSE,
           Drive_Fault_ACKN         := FALSE,
           Drive_F_Setpoint         := 5.000000e+01,
           Drive_in_operation       := #Temp1,
           Drive_Fault_Active       := "M67.7",
           Drive_Alarm_Active       := #Temp3,
           Freno                    := #Temp4,
           Drive_F_Act              := #RTemp1);
END_FUNCTION

FUNCTION "Gestione finecorsa" : VOID	// FC 18
VERSION : 0.1
BEGIN
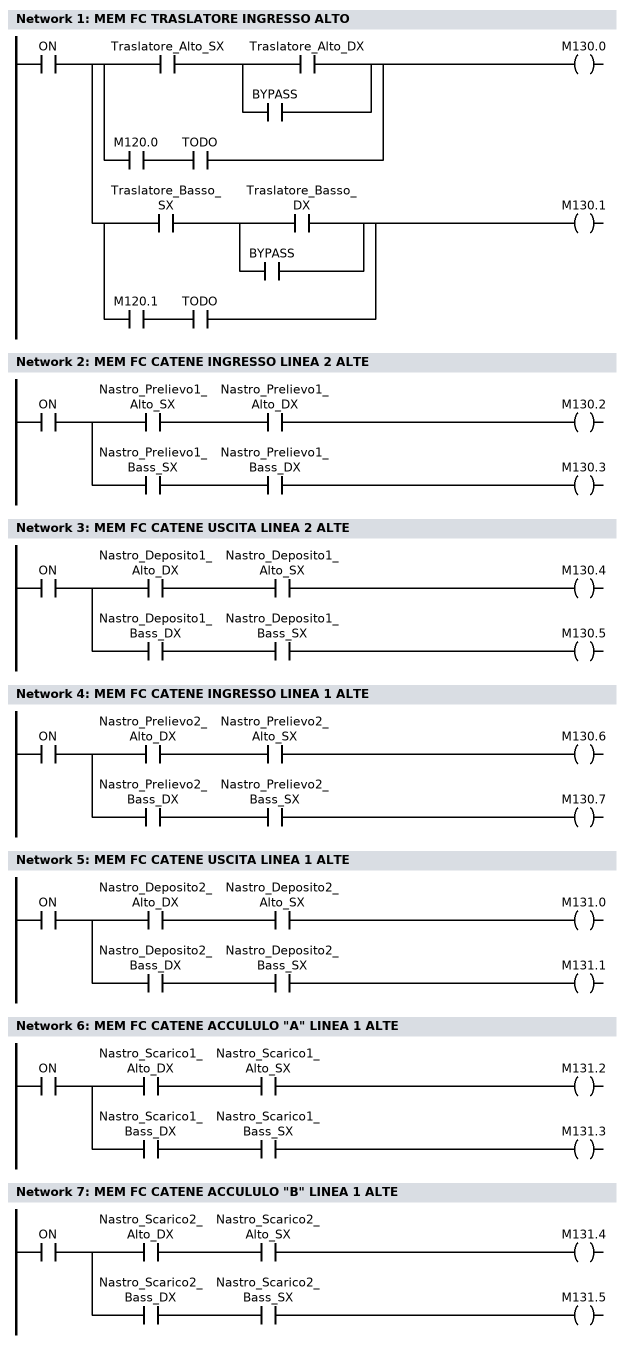
NETWORK
TITLE = MEM FC TRASLATORE INGRESSO ALTO
      A     "ON";
      =     L 0.0;
      A     L 0.0;
      A(;
      A     "Traslatore_Alto_SX";
      A(;
      O     "Traslatore_Alto_DX";
      O     "BYPASS";
      );
      O;
      A     "M120.0";
      A     "TODO";
      );
      =     "M130.0";
      A     L 0.0;
      A(;
      A     "Traslatore_Basso_SX";
      A(;
      O     "Traslatore_Basso_DX";
      O     "BYPASS";
      );
      O;
      A     "M120.1";
      A     "TODO";
      );
      =     "M130.1";
NETWORK
TITLE = MEM FC CATENE INGRESSO LINEA 2 ALTE
      A     "ON";
      =     L 0.0;
      A     L 0.0;
      A     "Nastro_Prelievo1_Alto_SX";
      A     "Nastro_Prelievo1_Alto_DX";
      =     "M130.2";
      A     L 0.0;
      A     "Nastro_Prelievo1_Bass_SX";
      A     "Nastro_Prelievo1_Bass_DX";
      =     "M130.3";
NETWORK
TITLE = MEM FC CATENE USCITA LINEA 2 ALTE
      A     "ON";
      =     L 0.0;
      A     L 0.0;
      A     "Nastro_Deposito1_Alto_DX";
      A     "Nastro_Deposito1_Alto_SX";
      =     "M130.4";
      A     L 0.0;
      A     "Nastro_Deposito1_Bass_DX";
      A     "Nastro_Deposito1_Bass_SX";
      =     "M130.5";
NETWORK
TITLE = MEM FC CATENE INGRESSO LINEA 1 ALTE
      A     "ON";
      =     L 0.0;
      A     L 0.0;
      A     "Nastro_Prelievo2_Alto_DX";
      A     "Nastro_Prelievo2_Alto_SX";
      =     "M130.6";
      A     L 0.0;
      A     "Nastro_Prelievo2_Bass_DX";
      A     "Nastro_Prelievo2_Bass_SX";
      =     "M130.7";
NETWORK
TITLE = MEM FC CATENE USCITA LINEA 1 ALTE
      A     "ON";
      =     L 0.0;
      A     L 0.0;
      A     "Nastro_Deposito2_Alto_DX";
      A     "Nastro_Deposito2_Alto_SX";
      =     "M131.0";
      A     L 0.0;
      A     "Nastro_Deposito2_Bass_DX";
      A     "Nastro_Deposito2_Bass_SX";
      =     "M131.1";
NETWORK
TITLE = MEM FC CATENE ACCULULO "A" LINEA 1 ALTE
      A     "ON";
      =     L 0.0;
      A     L 0.0;
      A     "Nastro_Scarico1_Alto_DX";
      A     "Nastro_Scarico1_Alto_SX";
      =     "M131.2";
      A     L 0.0;
      A     "Nastro_Scarico1_Bass_DX";
      A     "Nastro_Scarico1_Bass_SX";
      =     "M131.3";
NETWORK
TITLE = MEM FC CATENE ACCULULO "B" LINEA 1 ALTE
      A     "ON";
      =     L 0.0;
      A     L 0.0;
      A     "Nastro_Scarico2_Alto_DX";
      A     "Nastro_Scarico2_Alto_SX";
      =     "M131.4";
      A     L 0.0;
      A     "Nastro_Scarico2_Bass_DX";
      A     "Nastro_Scarico2_Bass_SX";
      =     "M131.5";
END_FUNCTION

FUNCTION "Gestione OP" : VOID	// FC 20
VERSION : 0.1
BEGIN
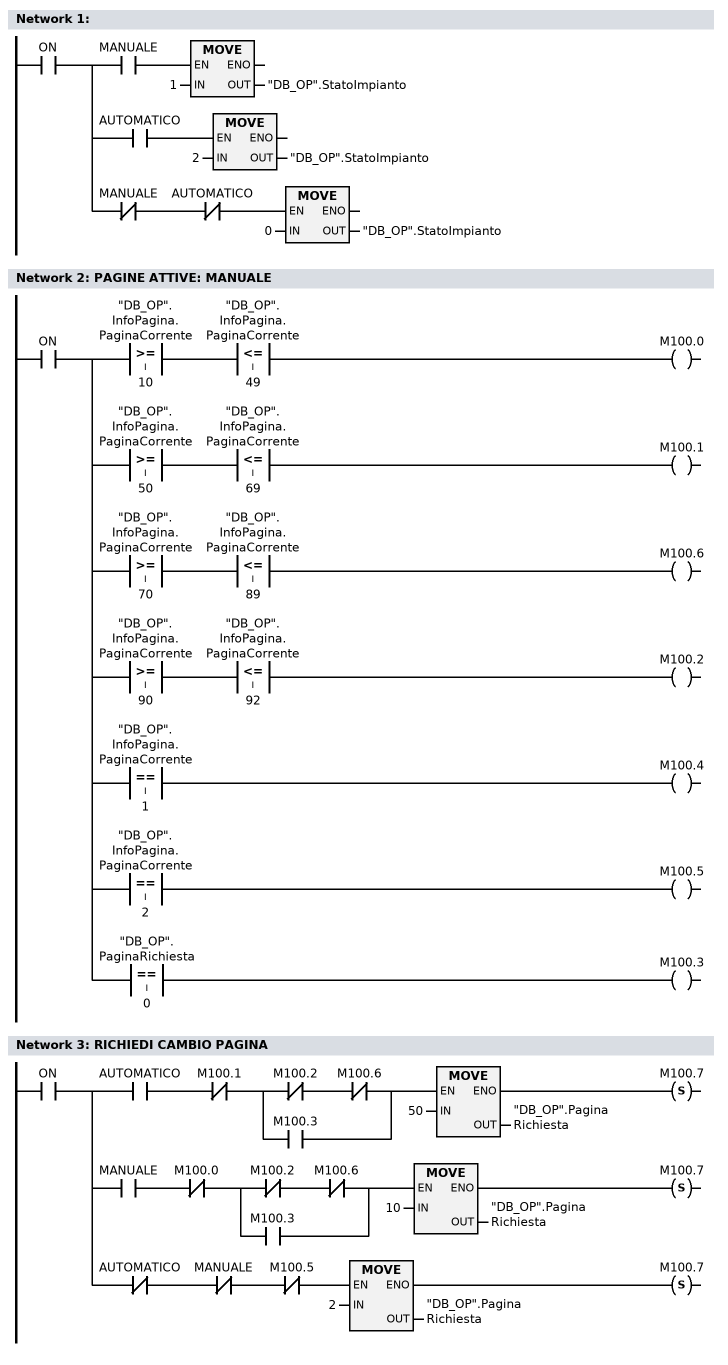
NETWORK
TITLE =
      A     "ON";
      =     L 0.0;
      A     L 0.0;
      A     "MANUALE";
      JNB   _001;
      L     1;
      T     "DB_OP".StatoImpianto;
_001: NOP   0;
      A     L 0.0;
      A     "AUTOMATICO";
      JNB   _002;
      L     2;
      T     "DB_OP".StatoImpianto;
_002: NOP   0;
      A     L 0.0;
      AN    "MANUALE";
      AN    "AUTOMATICO";
      JNB   _003;
      L     0;
      T     "DB_OP".StatoImpianto;
_003: NOP   0;
NETWORK
TITLE = PAGINE ATTIVE: MANUALE
      A     "ON";
      =     L 0.0;
      A     L 0.0;
      A(;
      L     "DB_OP".InfoPagina.PaginaCorrente;
      L     10;
      >=I;
      );
      A(;
      L     "DB_OP".InfoPagina.PaginaCorrente;
      L     49;
      <=I;
      );
      =     "M100.0";
      A     L 0.0;
      A(;
      L     "DB_OP".InfoPagina.PaginaCorrente;
      L     50;
      >=I;
      );
      A(;
      L     "DB_OP".InfoPagina.PaginaCorrente;
      L     69;
      <=I;
      );
      =     "M100.1";
      A     L 0.0;
      A(;
      L     "DB_OP".InfoPagina.PaginaCorrente;
      L     70;
      >=I;
      );
      A(;
      L     "DB_OP".InfoPagina.PaginaCorrente;
      L     89;
      <=I;
      );
      =     "M100.6";
      A     L 0.0;
      A(;
      L     "DB_OP".InfoPagina.PaginaCorrente;
      L     90;
      >=I;
      );
      A(;
      L     "DB_OP".InfoPagina.PaginaCorrente;
      L     92;
      <=I;
      );
      =     "M100.2";
      A     L 0.0;
      A(;
      L     "DB_OP".InfoPagina.PaginaCorrente;
      L     1;
      ==I;
      );
      =     "M100.4";
      A     L 0.0;
      A(;
      L     "DB_OP".InfoPagina.PaginaCorrente;
      L     2;
      ==I;
      );
      =     "M100.5";
      A     L 0.0;
      A(;
      L     "DB_OP".PaginaRichiesta;
      L     0;
      ==I;
      );
      =     "M100.3";
NETWORK
TITLE = RICHIEDI CAMBIO PAGINA
      A     "ON";
      =     L 0.0;
      A     L 0.0;
      A     "AUTOMATICO";
      AN    "M100.1";
      A(;
      AN    "M100.2";
      AN    "M100.6";
      O     "M100.3";
      );
      JNB   _004;
      L     50;
      T     "DB_OP".PaginaRichiesta;
      SET;
      SAVE;
      CLR;
_004: A     BR;
      S     "M100.7";
      A     L 0.0;
      A     "MANUALE";
      AN    "M100.0";
      A(;
      AN    "M100.2";
      AN    "M100.6";
      O     "M100.3";
      );
      JNB   _005;
      L     10;
      T     "DB_OP".PaginaRichiesta;
      SET;
      SAVE;
      CLR;
_005: A     BR;
      S     "M100.7";
      A     L 0.0;
      AN    "AUTOMATICO";
      AN    "MANUALE";
      AN    "M100.5";
      JNB   _006;
      L     2;
      T     "DB_OP".PaginaRichiesta;
      SET;
      SAVE;
      CLR;
_006: A     BR;
      S     "M100.7";
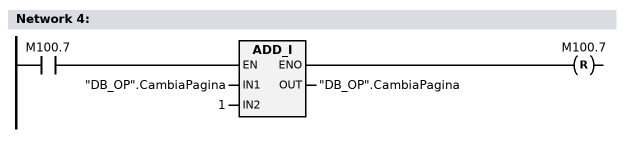
NETWORK
TITLE =
      A     "M100.7";
      JNB   _007;
      L     "DB_OP".CambiaPagina;
      L     1;
      +I;
      T     "DB_OP".CambiaPagina;
      AN    OV;
      SAVE;
      CLR;
_007: A     BR;
      R     "M100.7";
END_FUNCTION

FUNCTION "Gestione Timer e Counter" : VOID	// FC 30
VERSION : 0.1
BEGIN
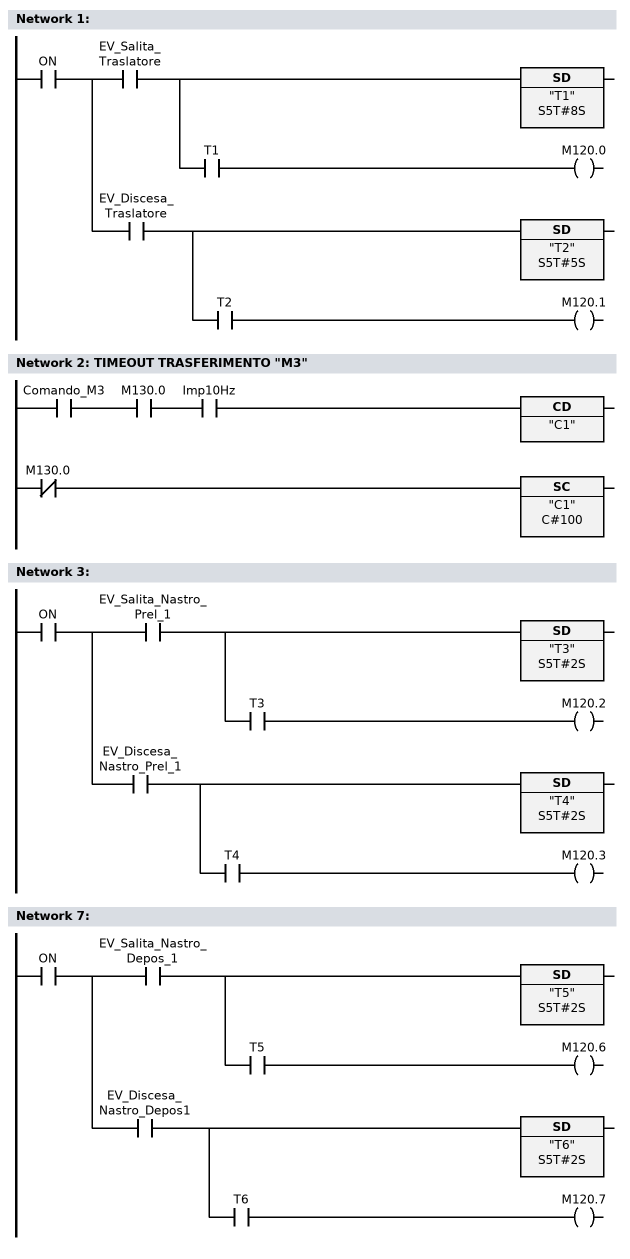
NETWORK
TITLE =
      A     "ON";
      =     L 0.0;
      A     L 0.0;
      A     "EV_Salita_Traslatore";
      =     L 0.1;
      A     L 0.1;
      BLD   102;
      L     S5T#8S;
      SD    "T1";
      A     L 0.1;
      A     "T1";
      =     "M120.0";
      A     L 0.0;
      A     "EV_Discesa_Traslatore";
      =     L 0.1;
      A     L 0.1;
      BLD   102;
      L     S5T#5S;
      SD    "T2";
      A     L 0.1;
      A     "T2";
      =     "M120.1";
NETWORK
TITLE = TIMEOUT TRASFERIMENTO "M3"
      A     "Comando_M3";
      A     "M130.0";
      A     "Imp10Hz";
      CD    "C1";
      BLD   101;
      AN    "M130.0";
      L     C#100;
      S     "C1";
      NOP   0;
      NOP   0;
      NOP   0;
      NOP   0;
NETWORK
TITLE =
      A     "ON";
      =     L 0.0;
      A     L 0.0;
      A     "EV_Salita_Nastro_Prel_1";
      =     L 0.1;
      A     L 0.1;
      BLD   102;
      L     S5T#2S;
      SD    "T3";
      A     L 0.1;
      A     "T3";
      =     "M120.2";
      A     L 0.0;
      A     "EV_Discesa_Nastro_Prel_1";
      =     L 0.1;
      A     L 0.1;
      BLD   102;
      L     S5T#2S;
      SD    "T4";
      A     L 0.1;
      A     "T4";
      =     "M120.3";
NETWORK
TITLE = TEMPO SVUOTAMENTO CATENA INGRESSO CADENZATORE LINEA 2
      A(;
      A     "M21.0";
      A     "Comando_M4";
      A     "Imp10Hz";
      CD    "C2";
      BLD   101;
      AN    "M21.0";
      A     "M120.4";
      L     C#60;
      S     "C2";
      NOP   0;
      NOP   0;
      NOP   0;
      A     "C2";
      );
      NOT;
      =     "M120.4";
NETWORK
TITLE = TEMPO SVUOTAMENTO CATENA INGRESSO CADENZATORE LINEA 2
      A(;
      A     "M20.4";
      A     "Comando_M4";
      A     "M130.2";
      A     "Imp10Hz";
      CD    "C20";
      BLD   101;
      AN    "M20.4";
      L     C#30;
      S     "C20";
      NOP   0;
      NOP   0;
      NOP   0;
      A     "C20";
      );
      NOT;
      =     "M122.5";
NETWORK
TITLE = TEMPO PASSO CATENE LINEA 2
      A(;
      A     "M21.3";
      A     "Comando_M5";
      A     "Imp10Hz";
      CD    "C3";
      BLD   101;
      AN    "M21.3";
      A     "M120.5";
      L     C#8;
      S     "C3";
      NOP   0;
      NOP   0;
      NOP   0;
      A     "C3";
      );
      NOT;
      =     "M120.5";
NETWORK
TITLE =
      A     "ON";
      =     L 0.0;
      A     L 0.0;
      A     "EV_Salita_Nastro_Depos_1";
      =     L 0.1;
      A     L 0.1;
      BLD   102;
      L     S5T#2S;
      SD    "T5";
      A     L 0.1;
      A     "T5";
      =     "M120.6";
      A     L 0.0;
      A     "EV_Discesa_Nastro_Depos1";
      =     L 0.1;
      A     L 0.1;
      BLD   102;
      L     S5T#2S;
      SD    "T6";
      A     L 0.1;
      A     "T6";
      =     "M120.7";
NETWORK
TITLE = TEMPO PASSO CATENE LINEA 2
      A(;
      A     "M24.6";
      A     "Comando_M17";
      A     "Imp10Hz";
      CD    "C4";
      BLD   101;
      AN    "M24.6";
      A     "M121.0";
      L     C#10;
      S     "C4";
      NOP   0;
      NOP   0;
      NOP   0;
      A     "C4";
      );
      NOT;
      =     "M121.0";
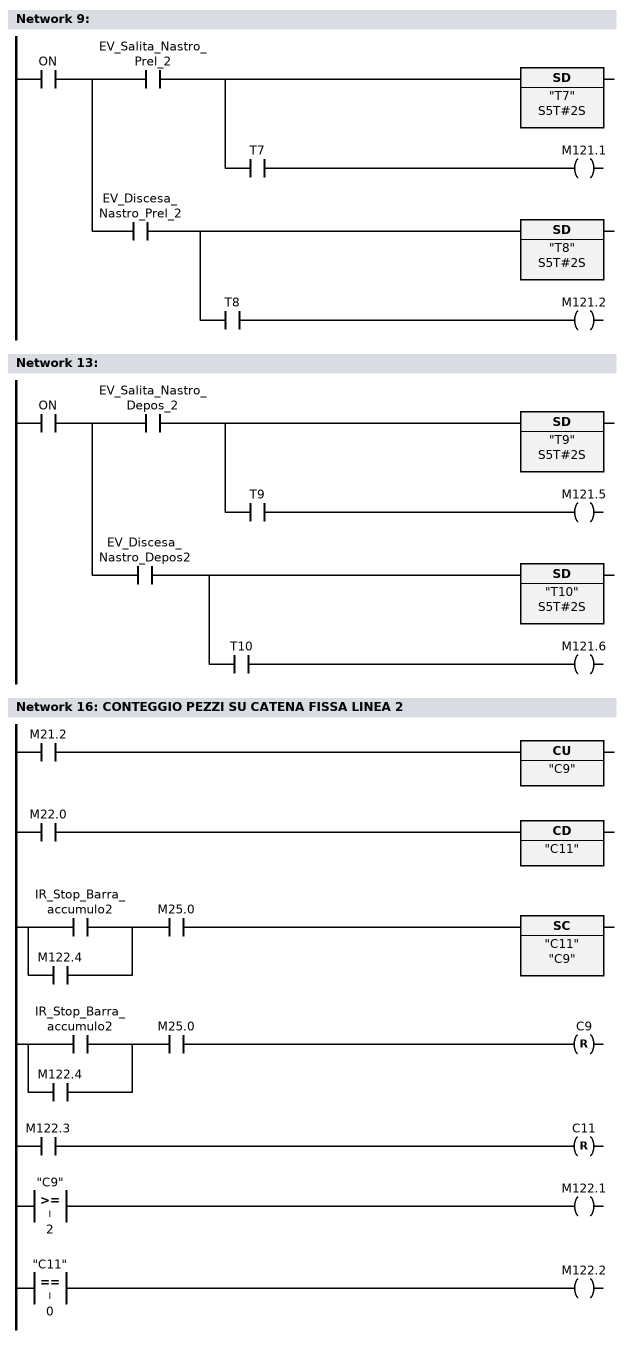
NETWORK
TITLE =
      A     "ON";
      =     L 0.0;
      A     L 0.0;
      A     "EV_Salita_Nastro_Prel_2";
      =     L 0.1;
      A     L 0.1;
      BLD   102;
      L     S5T#2S;
      SD    "T7";
      A     L 0.1;
      A     "T7";
      =     "M121.1";
      A     L 0.0;
      A     "EV_Discesa_Nastro_Prel_2";
      =     L 0.1;
      A     L 0.1;
      BLD   102;
      L     S5T#2S;
      SD    "T8";
      A     L 0.1;
      A     "T8";
      =     "M121.2";
NETWORK
TITLE = TEMPO SVUOTAMENTO CATENA INGRESSO CADENZATORE LINEA 1
      A(;
      A     "M41.0";
      A     "Comando_M11";
      A     "Imp10Hz";
      CD    "C5";
      BLD   101;
      AN    "M41.0";
      A     "M121.3";
      L     C#60;
      S     "C5";
      NOP   0;
      NOP   0;
      NOP   0;
      A     "C5";
      );
      NOT;
      =     "M121.3";
NETWORK
TITLE = RITARDO FUORI INGOMBRO M24
      A(;
      A     "M40.4";
      A     "Comando_M11";
      A     "M130.6";
      A     "Imp10Hz";
      CD    "C21";
      BLD   101;
      AN    "M40.4";
      L     C#30;
      S     "C21";
      NOP   0;
      NOP   0;
      NOP   0;
      A     "C21";
      );
      NOT;
      =     "M122.6";
NETWORK
TITLE = TEMPO PASSO CATENE LINEA 1
      A(;
      A     "M41.3";
      A     "Comando_M10";
      A     "Imp10Hz";
      CD    "C6";
      BLD   101;
      AN    "M41.3";
      A     "M121.4";
      L     C#8;
      S     "C6";
      NOP   0;
      NOP   0;
      NOP   0;
      A     "C6";
      );
      NOT;
      =     "M121.4";
NETWORK
TITLE =
      A     "ON";
      =     L 0.0;
      A     L 0.0;
      A     "EV_Salita_Nastro_Depos_2";
      =     L 0.1;
      A     L 0.1;
      BLD   102;
      L     S5T#2S;
      SD    "T9";
      A     L 0.1;
      A     "T9";
      =     "M121.5";
      A     L 0.0;
      A     "EV_Discesa_Nastro_Depos2";
      =     L 0.1;
      A     L 0.1;
      BLD   102;
      L     S5T#2S;
      SD    "T10";
      A     L 0.1;
      A     "T10";
      =     "M121.6";
NETWORK
TITLE =
      A(;
      A     "M21.1";
      AN    "Proximity_0_Cadenzatore1";
      A     "Comando_M7";
      A     "Imp10Hz";
      CD    "C7";
      BLD   101;
      A     "Proximity_0_Cadenzatore1";
      A     "M121.7";
      L     C#25;
      S     "C7";
      NOP   0;
      NOP   0;
      NOP   0;
      A     "C7";
      );
      NOT;
      =     "M121.7";
NETWORK
TITLE =
      A(;
      A     "M41.1";
      AN    "Proximity_0_Cadenzatore2";
      A     "Comando_M8";
      A     "Imp10Hz";
      CD    "C8";
      BLD   101;
      A     "Proximity_0_Cadenzatore2";
      A     "M122.0";
      L     C#25;
      S     "C8";
      NOP   0;
      NOP   0;
      NOP   0;
      A     "C8";
      );
      NOT;
      =     "M122.0";
NETWORK
TITLE = CONTEGGIO PEZZI SU CATENA FISSA LINEA 2
      A     "M21.2";
      CU    "C9";
      A     "M22.0";
      CD    "C11";
      A(;
      A     "IR_Stop_Barra_accumulo2";
      O     "M122.4";
      );
      A     "M25.0";
      L     "C9";
      S     "C11";
      A(;
      A     "IR_Stop_Barra_accumulo2";
      O     "M122.4";
      );
      A     "M25.0";
      R     "C9";
      A     "M122.3";
      R     "C11";
      L     "C9";
      L     2;
      >=I;
      =     "M122.1";
      L     "C11";
      L     0;
      ==I;
      =     "M122.2";
NETWORK
TITLE =
      A(;
      AN    "M25.0";
      A     "Comando_M6";
      A     "Imp10Hz";
      CD    "C10";
      BLD   101;
      A     "M25.0";
      L     C#60;
      S     "C10";
      NOP   0;
      NOP   0;
      NOP   0;
      A     "C10";
      );
      NOT;
      =     "M122.3";
NETWORK
TITLE =
      A(;
      A     "M25.0";
      A     "Comando_M6";
      A     "Imp10Hz";
      CD    "C12";
      BLD   101;
      AN    "M25.0";
      L     C#80;
      S     "C12";
      NOP   0;
      NOP   0;
      NOP   0;
      A     "C12";
      );
      NOT;
      =     "M122.4";
